LIN {X 0.078,Y -147.268,Z 1124.913,A 0.000,B 0.000,C 90.000,E1 164.393} C_DIS
LIN {X -0.047,Y -150.585,Z 1124.888,A 0.000,B 0.000,C 90.000,E1 159.880} C_DIS
LIN {X 0.032,Y -154.056,Z 1124.868,A 0.000,B 0.000,C 90.000,E1 156.230} C_DIS
LIN {X -0.042,Y -157.475,Z 1124.848,A 0.000,B 0.000,C 90.000,E1 152.666} C_DIS
LIN {X 0.044,Y -161.698,Z 1124.828,A 0.000,B 0.000,C 90.000,E1 149.076} C_DIS
LIN {X -0.078,Y -165.893,Z 1124.809,A 0.000,B 0.000,C 90.000,E1 145.595} C_DIS
LIN {X 0.047,Y -170.875,Z 1124.789,A 0.000,B 0.000,C 90.000,E1 142.065} C_DIS
LIN {X 0.075,Y -175.743,Z 1124.770,A 0.000,B 0.000,C 90.000,E1 138.609} C_DIS
LIN {X -0.052,Y -181.354,Z 1124.751,A 0.000,B 0.000,C 90.000,E1 135.243} C_DIS
LIN {X 0.081,Y -186.844,Z 1124.733,A 0.000,B 0.000,C 90.000,E1 131.838} C_DIS
LIN {X 0.035,Y -191.431,Z 1124.719,A 0.000,B 0.000,C 90.000,E1 129.358} C_DIS
LIN {X -0.032,Y -197.282,Z 1124.700,A 0.000,B 0.000,C 90.000,E1 126.091} C_DIS
LIN {X 0.094,Y -200.751,Z 1124.691,A 0.000,B 0.000,C 90.000,E1 124.326} C_DIS
LIN {X 0.093,Y -309.580,Z 1124.691,A 0.000,B 0.000,C 90.000,E1 124.326} C_DIS
LIN {X -0.009,Y -310.783,Z 1124.691,A 0.000,B 0.000,C 90.000,E1 124.326} C_DIS
LIN {X 0.192,Y -314.940,Z 1124.690,A 0.000,B 0.000,C 90.000,E1 124.119} C_DIS
LIN {X -0.044,Y -317.242,Z 1124.689,A 0.000,B 0.000,C 90.000,E1 123.992} C_DIS
LIN {X -0.078,Y -320.395,Z 1124.687,A 0.000,B 0.000,C 90.000,E1 123.658} C_DIS
LIN {X -0.134,Y -322.373,Z 1124.685,A 0.000,B 0.000,C 90.000,E1 123.372} C_DIS
LIN {X 0.082,Y -323.924,Z 1124.684,A 0.000,B 0.000,C 90.000,E1 123.038} C_DIS
LIN {X -0.010,Y -326.368,Z 1124.680,A 0.000,B 0.000,C 90.000,E1 122.418} C_DIS
LIN {X 0.001,Y -337.171,Z 1124.664,A 0.000,B 0.000,C 90.000,E1 119.589} C_DIS
LIN {X -0.050,Y -349.350,Z 1124.649,A 0.000,B 0.000,C 90.000,E1 116.821} C_DIS
LIN {X 0.109,Y -363.007,Z 1124.634,A 0.000,B 0.000,C 90.000,E1 114.079} C_DIS
LIN {X 0.104,Y -376.488,Z 1124.621,A 0.000,B 0.000,C 90.000,E1 111.716} C_DIS
LIN {X 0.164,Y -391.330,Z 1124.608,A 0.000,B 0.000,C 90.000,E1 109.396} C_DIS
LIN {X -0.034,Y -407.636,Z 1124.595,A 0.000,B 0.000,C 90.000,E1 107.166} C_DIS
LIN {X 0.043,Y -425.524,Z 1124.583,A 0.000,B 0.000,C 90.000,E1 104.954} C_DIS
LIN {X 0.016,Y -444.998,Z 1124.571,A 0.000,B 0.000,C 90.000,E1 102.827} C_DIS
LIN {X 0.148,Y -465.243,Z 1124.560,A 0.000,B 0.000,C 90.000,E1 100.838} C_DIS
LIN {X 0.147,Y -467.826,Z 1124.559,A 0.000,B 0.000,C 90.000,E1 100.602} C_DIS
LIN {X 0.183,Y -470.038,Z 1124.558,A 0.000,B 0.000,C 90.000,E1 100.366} C_DIS
LIN {X 0.135,Y -471.709,Z 1124.556,A 0.000,B 0.000,C 90.000,E1 100.141} C_DIS
LIN {X -0.008,Y -473.101,Z 1124.555,A 0.000,B 0.000,C 90.000,E1 99.905} C_DIS
LIN {X -0.154,Y -474.134,Z 1124.554,A 0.000,B 0.000,C 90.000,E1 99.670} C_DIS
LIN {X -0.038,Y -475.327,Z 1124.551,A 0.000,B 0.000,C 90.000,E1 99.151} C_DIS
LIN {X 0.158,Y -475.518,Z 1124.548,A 0.000,B 0.000,C 90.000,E1 98.624} C_DIS
LIN {X -0.181,Y -474.740,Z 1124.545,A 0.000,B 0.000,C 90.000,E1 98.163} C_DIS
LIN {X -0.048,Y -472.867,Z 1124.542,A 0.000,B 0.000,C 90.000,E1 97.644} C_DIS
LIN {X -0.186,Y -471.408,Z 1124.541,A 0.000,B 0.000,C 90.000,E1 97.409} C_DIS
LIN {X -0.064,Y -455.155,Z 1124.528,A 0.000,B 0.000,C 90.000,E1 95.106} C_DIS
LIN {X -0.132,Y -441.016,Z 1124.517,A 0.000,B 0.000,C 90.000,E1 93.037} C_DIS
LIN {X 0.012,Y -426.343,Z 1124.504,A 0.000,B 0.000,C 90.000,E1 90.630} C_DIS
LIN {X 0.187,Y -412.584,Z 1124.490,A 0.000,B 0.000,C 90.000,E1 88.167} C_DIS
LIN {X -0.140,Y -403.696,Z 1124.481,A 0.000,B 0.000,C 90.000,E1 86.560} C_DIS
LIN {X -0.185,Y -393.159,Z 1124.470,A 0.000,B 0.000,C 90.000,E1 84.609} C_DIS
LIN {X 0.011,Y -382.701,Z 1124.459,A 0.000,B 0.000,C 90.000,E1 82.591} C_DIS
LIN {X 0.081,Y -373.658,Z 1124.449,A 0.000,B 0.000,C 90.000,E1 80.849} C_DIS
LIN {X -0.009,Y -364.263,Z 1124.439,A 0.000,B 0.000,C 90.000,E1 79.106} C_DIS
LIN {X -0.200,Y -354.498,Z 1124.430,A 0.000,B 0.000,C 90.000,E1 77.353} C_DIS
LIN {X -0.144,Y -342.981,Z 1124.418,A 0.000,B 0.000,C 90.000,E1 75.227} C_DIS
LIN {X 0.050,Y -329.902,Z 1124.404,A 0.000,B 0.000,C 90.000,E1 72.725} C_DIS
LIN {X -0.017,Y -314.350,Z 1124.386,A 0.000,B 0.000,C 90.000,E1 69.571} C_DIS
LIN {X 0.067,Y -299.831,Z 1124.368,A 0.000,B 0.000,C 90.000,E1 66.305} C_DIS
LIN {X 0.084,Y -288.803,Z 1124.354,A 0.000,B 0.000,C 90.000,E1 63.640} C_DIS
LIN {X 0.089,Y -278.065,Z 1124.339,A 0.000,B 0.000,C 90.000,E1 60.923} C_DIS
LIN {X -0.064,Y -269.002,Z 1124.325,A 0.000,B 0.000,C 90.000,E1 58.535} C_DIS
LIN {X 0.071,Y -256.550,Z 1124.306,A 0.000,B 0.000,C 90.000,E1 54.975} C_DIS
LIN {X -0.011,Y -245.997,Z 1124.287,A 0.000,B 0.000,C 90.000,E1 51.743} C_DIS
LIN {X 0.089,Y -236.309,Z 1124.269,A 0.000,B 0.000,C 90.000,E1 48.405} C_DIS
LIN {X 0.096,Y -228.271,Z 1124.252,A 0.000,B 0.000,C 90.000,E1 45.405} C_DIS
LIN {X 0.063,Y -220.623,Z 1124.235,A 0.000,B 0.000,C 90.000,E1 42.366} C_DIS
LIN {X 0.036,Y -213.340,Z 1124.218,A 0.000,B 0.000,C 90.000,E1 39.277} C_DIS
LIN {X 0.023,Y -206.482,Z 1124.201,A 0.000,B 0.000,C 90.000,E1 36.137} C_DIS
LIN {X -0.021,Y -200.095,Z 1124.183,A 0.000,B 0.000,C 90.000,E1 32.959} C_DIS
LIN {X -0.089,Y -194.301,Z 1124.165,A 0.000,B 0.000,C 90.000,E1 29.745} C_DIS
LIN {X 0.018,Y -189.100,Z 1124.147,A 0.000,B 0.000,C 90.000,E1 26.437} C_DIS
LIN {X -0.007,Y -184.527,Z 1124.129,A 0.000,B 0.000,C 90.000,E1 23.131} C_DIS
LIN {X -0.066,Y -179.757,Z 1124.105,A 0.000,B 0.000,C 90.000,E1 18.960} C_DIS
LIN {X -0.036,Y -175.995,Z 1124.082,A 0.000,B 0.000,C 90.000,E1 14.717} C_DIS
LIN {X 0.069,Y -172.856,Z 1124.053,A 0.000,B 0.000,C 90.000,E1 9.557} C_DIS
LIN {X -0.002,Y -170.940,Z 1124.010,A 0.000,B 0.000,C 90.000,E1 1.835} C_DIS
LIN {X -0.050,Y -172.525,Z 1123.964,A 0.000,B 0.000,C 90.000,E1 353.514} C_DIS
LIN {X 0.020,Y -175.335,Z 1123.935,A 0.000,B 0.000,C 90.000,E1 348.342} C_DIS
LIN {X -0.052,Y -178.751,Z 1123.912,A 0.000,B 0.000,C 90.000,E1 344.102} C_DIS
LIN {X -0.072,Y -183.004,Z 1123.888,A 0.000,B 0.000,C 90.000,E1 339.880} C_DIS
LIN {X 0.066,Y -187.097,Z 1123.870,A 0.000,B 0.000,C 90.000,E1 336.485} C_DIS
LIN {X 0.023,Y -191.887,Z 1123.851,A 0.000,B 0.000,C 90.000,E1 333.179} C_DIS
LIN {X -0.066,Y -197.332,Z 1123.833,A 0.000,B 0.000,C 90.000,E1 329.921} C_DIS
LIN {X 0.107,Y -203.385,Z 1123.815,A 0.000,B 0.000,C 90.000,E1 326.628} C_DIS
LIN {X -0.018,Y -210.290,Z 1123.797,A 0.000,B 0.000,C 90.000,E1 323.463} C_DIS
LIN {X 0.116,Y -217.935,Z 1123.779,A 0.000,B 0.000,C 90.000,E1 320.275} C_DIS
LIN {X -0.067,Y -226.470,Z 1123.762,A 0.000,B 0.000,C 90.000,E1 317.229} C_DIS
LIN {X -0.061,Y -236.018,Z 1123.745,A 0.000,B 0.000,C 90.000,E1 314.190} C_DIS
LIN {X 0.073,Y -243.903,Z 1123.733,A 0.000,B 0.000,C 90.000,E1 311.919} C_DIS
LIN {X 0.075,Y -255.655,Z 1123.717,A 0.000,B 0.000,C 90.000,E1 308.991} C_DIS
LIN {X -0.061,Y -265.510,Z 1123.705,A 0.000,B 0.000,C 90.000,E1 306.870} C_DIS
LIN {X 0.065,Y -279.774,Z 1123.689,A 0.000,B 0.000,C 90.000,E1 304.040} C_DIS
LIN {X -0.065,Y -294.990,Z 1123.674,A 0.000,B 0.000,C 90.000,E1 301.337} C_DIS
LIN {X -0.059,Y -314.165,Z 1123.657,A 0.000,B 0.000,C 90.000,E1 298.359} C_DIS
LIN {X -0.007,Y -330.283,Z 1123.645,A 0.000,B 0.000,C 90.000,E1 296.104} C_DIS
LIN {X -0.108,Y -345.206,Z 1123.635,A 0.000,B 0.000,C 90.000,E1 294.259} C_DIS
LIN {X 0.181,Y -358.205,Z 1123.627,A 0.000,B 0.000,C 90.000,E1 292.770} C_DIS
LIN {X -0.036,Y -371.604,Z 1123.619,A 0.000,B 0.000,C 90.000,E1 291.461} C_DIS
LIN {X -0.066,Y -393.675,Z 1123.608,A 0.000,B 0.000,C 90.000,E1 289.450} C_DIS
LIN {X -0.014,Y -404.411,Z 1123.603,A 0.000,B 0.000,C 90.000,E1 288.489} C_DIS
LIN {X -0.010,Y -414.928,Z 1123.597,A 0.000,B 0.000,C 90.000,E1 287.511} C_DIS
LIN {X 0.218,Y -422.666,Z 1123.593,A 0.000,B 0.000,C 90.000,E1 286.732} C_DIS
LIN {X -0.221,Y -430.176,Z 1123.589,A 0.000,B 0.000,C 90.000,E1 286.024} C_DIS
LIN {X 0.112,Y -437.408,Z 1123.584,A 0.000,B 0.000,C 90.000,E1 285.190} C_DIS
LIN {X -0.030,Y -444.251,Z 1123.580,A 0.000,B 0.000,C 90.000,E1 284.411} C_DIS
LIN {X 0.216,Y -450.480,Z 1123.576,A 0.000,B 0.000,C 90.000,E1 283.592} C_DIS
LIN {X -0.174,Y -454.313,Z 1123.573,A 0.000,B 0.000,C 90.000,E1 283.119} C_DIS
LIN {X 0.165,Y -459.376,Z 1123.568,A 0.000,B 0.000,C 90.000,E1 282.299} C_DIS
LIN {X 0.107,Y -463.742,Z 1123.564,A 0.000,B 0.000,C 90.000,E1 281.535} C_DIS
LIN {X -0.159,Y -468.724,Z 1123.558,A 0.000,B 0.000,C 90.000,E1 280.546} C_DIS
LIN {X -0.147,Y -471.821,Z 1123.554,A 0.000,B 0.000,C 90.000,E1 279.782} C_DIS
LIN {X -0.053,Y -473.578,Z 1123.551,A 0.000,B 0.000,C 90.000,E1 279.265} C_DIS
LIN {X 0.057,Y -474.975,Z 1123.549,A 0.000,B 0.000,C 90.000,E1 278.746} C_DIS
LIN {X 0.249,Y -476.177,Z 1123.546,A 0.000,B 0.000,C 90.000,E1 278.219} C_DIS
LIN {X -0.093,Y -477.066,Z 1123.543,A 0.000,B 0.000,C 90.000,E1 277.757} C_DIS
LIN {X 0.046,Y -477.654,Z 1123.540,A 0.000,B 0.000,C 90.000,E1 277.239} C_DIS
LIN {X 0.191,Y -477.940,Z 1123.537,A 0.000,B 0.000,C 90.000,E1 276.720} C_DIS
LIN {X -0.135,Y -477.901,Z 1123.535,A 0.000,B 0.000,C 90.000,E1 276.258} C_DIS
LIN {X 0.015,Y -477.520,Z 1123.532,A 0.000,B 0.000,C 90.000,E1 275.739} C_DIS
LIN {X 0.163,Y -476.836,Z 1123.529,A 0.000,B 0.000,C 90.000,E1 275.220} C_DIS
LIN {X -0.167,Y -475.804,Z 1123.526,A 0.000,B 0.000,C 90.000,E1 274.759} C_DIS
LIN {X -0.063,Y -474.319,Z 1123.524,A 0.000,B 0.000,C 90.000,E1 274.245} C_DIS
LIN {X 0.069,Y -472.342,Z 1123.521,A 0.000,B 0.000,C 90.000,E1 273.726} C_DIS
LIN {X -0.119,Y -471.140,Z 1123.519,A 0.000,B 0.000,C 90.000,E1 273.498} C_DIS
LIN {X -0.007,Y -468.090,Z 1123.517,A 0.000,B 0.000,C 90.000,E1 272.980} C_DIS
LIN {X -0.202,Y -466.283,Z 1123.515,A 0.000,B 0.000,C 90.000,E1 272.751} C_DIS
LIN {X -0.140,Y -461.786,Z 1123.512,A 0.000,B 0.000,C 90.000,E1 272.236} C_DIS
LIN {X 0.111,Y -459.021,Z 1123.511,A 0.000,B 0.000,C 90.000,E1 271.949} C_DIS
LIN {X 0.029,Y -452.897,Z 1123.508,A 0.000,B 0.000,C 90.000,E1 271.489} C_DIS
LIN {X 0.040,Y -446.345,Z 1123.506,A 0.000,B 0.000,C 90.000,E1 271.088} C_DIS
LIN {X 0.084,Y -439.442,Z 1123.504,A 0.000,B 0.000,C 90.000,E1 270.745} C_DIS
LIN {X 0.121,Y -432.411,Z 1123.503,A 0.000,B 0.000,C 90.000,E1 270.458} C_DIS
LIN {X 0.079,Y -425.348,Z 1123.501,A 0.000,B 0.000,C 90.000,E1 270.229} C_DIS
LIN {X -0.107,Y -418.092,Z 1123.500,A 0.000,B 0.000,C 90.000,E1 270.057} C_DIS
LIN {X -0.044,Y -410.673,Z 1123.499,A 0.000,B 0.000,C 90.000,E1 269.885} C_DIS
LIN {X -0.162,Y -403.059,Z 1123.499,A 0.000,B 0.000,C 90.000,E1 269.771} C_DIS
LIN {X -0.080,Y -393.478,Z 1123.498,A 0.000,B 0.000,C 90.000,E1 269.656} C_DIS
LIN {X 0.007,Y -384.032,Z 1123.498,A 0.000,B 0.000,C 90.000,E1 269.599} C_DIS
LIN {X -0.019,Y -181.463,Z 1123.498,A 0.000,B 0.000,C 90.000,E1 269.599} C_DIS
LIN {X -0.068,Y -180.906,Z 1123.474,A 0.000,B 0.000,C 90.000,E1 265.355} C_DIS
LIN {X 0.006,Y -180.671,Z 1123.469,A 0.000,B 0.000,C 90.000,E1 264.489} C_DIS
LIN {X 0.080,Y -178.752,Z 1123.441,A 0.000,B 0.000,C 90.000,E1 259.398} C_DIS
LIN {X -0.022,Y -175.799,Z 1123.413,A 0.000,B 0.000,C 90.000,E1 254.338} C_DIS
LIN {X -0.028,Y -171.985,Z 1123.384,A 0.000,B 0.000,C 90.000,E1 249.209} C_DIS
LIN {X 0.010,Y -171.391,Z 1123.380,A 0.000,B 0.000,C 90.000,E1 248.337} C_DIS
LIN {X -0.004,Y -167.634,Z 1123.356,A 0.000,B 0.000,C 90.000,E1 244.024} C_DIS
LIN {X 0.010,Y -166.292,Z 1123.346,A 0.000,B 0.000,C 90.000,E1 242.281} C_DIS
LIN {X 0.004,Y -163.039,Z 1123.327,A 0.000,B 0.000,C 90.000,E1 238.791} C_DIS
LIN {X -0.034,Y -160.970,Z 1123.312,A 0.000,B 0.000,C 90.000,E1 236.167} C_DIS
LIN {X -0.056,Y -157.722,Z 1123.292,A 0.000,B 0.000,C 90.000,E1 232.637} C_DIS
LIN {X 0.103,Y -155.762,Z 1123.277,A 0.000,B 0.000,C 90.000,E1 229.908} C_DIS
LIN {X -0.060,Y -152.017,Z 1123.253,A 0.000,B 0.000,C 90.000,E1 225.486} C_DIS
LIN {X -0.043,Y -150.264,Z 1123.238,A 0.000,B 0.000,C 90.000,E1 222.771} C_DIS
LIN {X -0.024,Y -147.017,Z 1123.212,A 0.000,B 0.000,C 90.000,E1 218.222} C_DIS
LIN {X -0.003,Y -145.600,Z 1123.197,A 0.000,B 0.000,C 90.000,E1 215.471} C_DIS
LIN {X 0.001,Y -142.986,Z 1123.172,A 0.000,B 0.000,C 90.000,E1 210.875} C_DIS
LIN {X 0.000,Y -141.613,Z 1123.151,A 0.000,B 0.000,C 90.000,E1 207.180} C_DIS
LIN {X 0.042,Y -139.428,Z 1123.115,A 0.000,B 0.000,C 90.000,E1 200.663} C_DIS
LIN {X -0.038,Y -139.158,Z 1123.104,A 0.000,B 0.000,C 90.000,E1 198.833} C_DIS
LIN {X -0.022,Y -138.343,Z 1123.058,A 0.000,B 0.000,C 90.000,E1 190.423} C_DIS
LIN {X -0.039,Y -139.481,Z 1123.006,A 0.000,B 0.000,C 90.000,E1 181.088} C_DIS
LIN {X 0.041,Y -141.072,Z 1122.975,A 0.000,B 0.000,C 90.000,E1 175.469} C_DIS
LIN {X -0.004,Y -142.447,Z 1122.959,A 0.000,B 0.000,C 90.000,E1 172.704} C_DIS
LIN {X -0.056,Y -144.687,Z 1122.934,A 0.000,B 0.000,C 90.000,E1 168.105} C_DIS
LIN {X 0.039,Y -147.280,Z 1122.913,A 0.000,B 0.000,C 90.000,E1 164.393} C_DIS
LIN {X 0.054,Y -150.598,Z 1122.888,A 0.000,B 0.000,C 90.000,E1 159.826} C_DIS
LIN {X -0.009,Y -154.071,Z 1122.868,A 0.000,B 0.000,C 90.000,E1 156.230} C_DIS
LIN {X 0.057,Y -157.491,Z 1122.848,A 0.000,B 0.000,C 90.000,E1 152.615} C_DIS
LIN {X 0.003,Y -161.717,Z 1122.828,A 0.000,B 0.000,C 90.000,E1 149.076} C_DIS
LIN {X 0.017,Y -165.911,Z 1122.809,A 0.000,B 0.000,C 90.000,E1 145.548} C_DIS
LIN {X 0.004,Y -170.897,Z 1122.789,A 0.000,B 0.000,C 90.000,E1 142.065} C_DIS
LIN {X 0.030,Y -175.765,Z 1122.770,A 0.000,B 0.000,C 90.000,E1 138.609} C_DIS
LIN {X -0.097,Y -181.375,Z 1122.751,A 0.000,B 0.000,C 90.000,E1 135.243} C_DIS
LIN {X 0.036,Y -186.870,Z 1122.733,A 0.000,B 0.000,C 90.000,E1 131.838} C_DIS
LIN {X -0.011,Y -191.454,Z 1122.719,A 0.000,B 0.000,C 90.000,E1 129.358} C_DIS
LIN {X -0.079,Y -197.308,Z 1122.700,A 0.000,B 0.000,C 90.000,E1 126.091} C_DIS
LIN {X -0.073,Y -200.691,Z 1122.691,A 0.000,B 0.000,C 90.000,E1 124.405} C_DIS
LIN {X -0.165,Y -309.271,Z 1122.691,A 0.000,B 0.000,C 90.000,E1 124.405} C_DIS
LIN {X -0.054,Y -314.738,Z 1122.690,A 0.000,B 0.000,C 90.000,E1 124.199} C_DIS
LIN {X 0.059,Y -317.249,Z 1122.689,A 0.000,B 0.000,C 90.000,E1 123.992} C_DIS
LIN {X 0.024,Y -320.601,Z 1122.687,A 0.000,B 0.000,C 90.000,E1 123.627} C_DIS
LIN {X 0.202,Y -322.540,Z 1122.685,A 0.000,B 0.000,C 90.000,E1 123.293} C_DIS
LIN {X -0.066,Y -324.057,Z 1122.683,A 0.000,B 0.000,C 90.000,E1 123.038} C_DIS
LIN {X -0.128,Y -329.897,Z 1122.675,A 0.000,B 0.000,C 90.000,E1 121.465} C_DIS
LIN {X 0.100,Y -341.161,Z 1122.659,A 0.000,B 0.000,C 90.000,E1 118.615} C_DIS
LIN {X 0.176,Y -353.831,Z 1122.644,A 0.000,B 0.000,C 90.000,E1 115.848} C_DIS
LIN {X -0.176,Y -368.026,Z 1122.629,A 0.000,B 0.000,C 90.000,E1 113.206} C_DIS
LIN {X -0.068,Y -382.020,Z 1122.616,A 0.000,B 0.000,C 90.000,E1 110.844} C_DIS
LIN {X -0.012,Y -397.413,Z 1122.603,A 0.000,B 0.000,C 90.000,E1 108.544} C_DIS
LIN {X -0.074,Y -414.315,Z 1122.591,A 0.000,B 0.000,C 90.000,E1 106.315} C_DIS
LIN {X 0.045,Y -432.847,Z 1122.578,A 0.000,B 0.000,C 90.000,E1 104.120} C_DIS
LIN {X -0.125,Y -452.724,Z 1122.567,A 0.000,B 0.000,C 90.000,E1 102.063} C_DIS
LIN {X -0.017,Y -468.016,Z 1122.559,A 0.000,B 0.000,C 90.000,E1 100.602} C_DIS
LIN {X -0.007,Y -470.194,Z 1122.558,A 0.000,B 0.000,C 90.000,E1 100.366} C_DIS
LIN {X -0.082,Y -471.839,Z 1122.556,A 0.000,B 0.000,C 90.000,E1 100.141} C_DIS
LIN {X -0.226,Y -473.187,Z 1122.555,A 0.000,B 0.000,C 90.000,E1 99.905} C_DIS
LIN {X 0.096,Y -474.185,Z 1122.553,A 0.000,B 0.000,C 90.000,E1 99.613} C_DIS
LIN {X -0.256,Y -475.321,Z 1122.551,A 0.000,B 0.000,C 90.000,E1 99.151} C_DIS
LIN {X -0.060,Y -475.460,Z 1122.548,A 0.000,B 0.000,C 90.000,E1 98.624} C_DIS
LIN {X 0.072,Y -474.628,Z 1122.545,A 0.000,B 0.000,C 90.000,E1 98.106} C_DIS
LIN {X 0.204,Y -472.688,Z 1122.542,A 0.000,B 0.000,C 90.000,E1 97.587} C_DIS
LIN {X 0.065,Y -471.185,Z 1122.541,A 0.000,B 0.000,C 90.000,E1 97.352} C_DIS
LIN {X 0.175,Y -454.915,Z 1122.528,A 0.000,B 0.000,C 90.000,E1 95.049} C_DIS
LIN {X 0.095,Y -440.803,Z 1122.517,A 0.000,B 0.000,C 90.000,E1 92.980} C_DIS
LIN {X -0.200,Y -426.134,Z 1122.503,A 0.000,B 0.000,C 90.000,E1 90.630} C_DIS
LIN {X -0.010,Y -412.392,Z 1122.490,A 0.000,B 0.000,C 90.000,E1 88.165} C_DIS
LIN {X 0.054,Y -403.476,Z 1122.481,A 0.000,B 0.000,C 90.000,E1 86.502} C_DIS
LIN {X 0.037,Y -392.943,Z 1122.470,A 0.000,B 0.000,C 90.000,E1 84.546} C_DIS
LIN {X -0.196,Y -382.457,Z 1122.459,A 0.000,B 0.000,C 90.000,E1 82.591} C_DIS
LIN {X -0.125,Y -373.410,Z 1122.449,A 0.000,B 0.000,C 90.000,E1 80.849} C_DIS
LIN {X 0.143,Y -363.997,Z 1122.439,A 0.000,B 0.000,C 90.000,E1 79.050} C_DIS
LIN {X 0.020,Y -354.232,Z 1122.429,A 0.000,B 0.000,C 90.000,E1 77.285} C_DIS
LIN {X -0.016,Y -342.704,Z 1122.418,A 0.000,B 0.000,C 90.000,E1 75.172} C_DIS
LIN {X -0.153,Y -329.628,Z 1122.404,A 0.000,B 0.000,C 90.000,E1 72.725} C_DIS
LIN {X 0.076,Y -314.071,Z 1122.386,A 0.000,B 0.000,C 90.000,E1 69.518} C_DIS
LIN {X -0.023,Y -301.005,Z 1122.370,A 0.000,B 0.000,C 90.000,E1 66.613} C_DIS
LIN {X -0.114,Y -288.562,Z 1122.353,A 0.000,B 0.000,C 90.000,E1 63.640} C_DIS
LIN {X 0.090,Y -276.514,Z 1122.336,A 0.000,B 0.000,C 90.000,E1 60.539} C_DIS
LIN {X 0.037,Y -267.447,Z 1122.323,A 0.000,B 0.000,C 90.000,E1 58.122} C_DIS
LIN {X -0.123,Y -256.262,Z 1122.305,A 0.000,B 0.000,C 90.000,E1 54.975} C_DIS
LIN {X -0.012,Y -245.726,Z 1122.287,A 0.000,B 0.000,C 90.000,E1 51.698} C_DIS
LIN {X -0.111,Y -235.996,Z 1122.269,A 0.000,B 0.000,C 90.000,E1 48.405} C_DIS
LIN {X -0.106,Y -227.948,Z 1122.252,A 0.000,B 0.000,C 90.000,E1 45.405} C_DIS
LIN {X 0.023,Y -220.291,Z 1122.235,A 0.000,B 0.000,C 90.000,E1 42.324} C_DIS
LIN {X 0.131,Y -212.976,Z 1122.218,A 0.000,B 0.000,C 90.000,E1 39.197} C_DIS
LIN {X -0.017,Y -206.098,Z 1122.200,A 0.000,B 0.000,C 90.000,E1 36.091} C_DIS
LIN {X 0.046,Y -199.720,Z 1122.183,A 0.000,B 0.000,C 90.000,E1 32.880} C_DIS
LIN {X -0.036,Y -193.939,Z 1122.165,A 0.000,B 0.000,C 90.000,E1 29.667} C_DIS
LIN {X 0.056,Y -188.733,Z 1122.146,A 0.000,B 0.000,C 90.000,E1 26.360} C_DIS
LIN {X -0.056,Y -184.163,Z 1122.128,A 0.000,B 0.000,C 90.000,E1 23.078} C_DIS
LIN {X 0.020,Y -180.266,Z 1122.109,A 0.000,B 0.000,C 90.000,E1 19.704} C_DIS
LIN {X 0.000,Y -176.334,Z 1122.086,A 0.000,B 0.000,C 90.000,E1 15.481} C_DIS
LIN {X 0.087,Y -173.408,Z 1122.062,A 0.000,B 0.000,C 90.000,E1 11.186} C_DIS
LIN {X -0.060,Y -171.090,Z 1122.029,A 0.000,B 0.000,C 90.000,E1 5.220} C_DIS
LIN {X -0.062,Y -172.230,Z 1121.964,A 0.000,B 0.000,C 90.000,E1 353.514} C_DIS
LIN {X -0.004,Y -175.013,Z 1121.935,A 0.000,B 0.000,C 90.000,E1 348.342} C_DIS
LIN {X -0.086,Y -178.430,Z 1121.911,A 0.000,B 0.000,C 90.000,E1 344.102} C_DIS
LIN {X 0.055,Y -182.673,Z 1121.888,A 0.000,B 0.000,C 90.000,E1 339.826} C_DIS
LIN {X 0.011,Y -186.756,Z 1121.869,A 0.000,B 0.000,C 90.000,E1 336.485} C_DIS
LIN {X -0.040,Y -191.571,Z 1121.851,A 0.000,B 0.000,C 90.000,E1 333.179} C_DIS
LIN {X 0.030,Y -197.013,Z 1121.833,A 0.000,B 0.000,C 90.000,E1 329.871} C_DIS
LIN {X 0.022,Y -203.098,Z 1121.815,A 0.000,B 0.000,C 90.000,E1 326.628} C_DIS
LIN {X 0.056,Y -210.032,Z 1121.797,A 0.000,B 0.000,C 90.000,E1 323.417} C_DIS
LIN {X 0.012,Y -217.714,Z 1121.779,A 0.000,B 0.000,C 90.000,E1 320.275} C_DIS
LIN {X -0.015,Y -226.272,Z 1121.762,A 0.000,B 0.000,C 90.000,E1 317.187} C_DIS
LIN {X -0.062,Y -237.098,Z 1121.743,A 0.000,B 0.000,C 90.000,E1 313.785} C_DIS
LIN {X 0.080,Y -246.590,Z 1121.729,A 0.000,B 0.000,C 90.000,E1 311.148} C_DIS
LIN {X -0.066,Y -255.540,Z 1121.717,A 0.000,B 0.000,C 90.000,E1 308.991} C_DIS
LIN {X 0.062,Y -267.220,Z 1121.703,A 0.000,B 0.000,C 90.000,E1 306.457} C_DIS
LIN {X 0.192,Y -283.502,Z 1121.685,A 0.000,B 0.000,C 90.000,E1 303.293} C_DIS
LIN {X 0.176,Y -295.064,Z 1121.674,A 0.000,B 0.000,C 90.000,E1 301.258} C_DIS
LIN {X 0.045,Y -314.270,Z 1121.657,A 0.000,B 0.000,C 90.000,E1 298.309} C_DIS
LIN {X 0.110,Y -330.421,Z 1121.645,A 0.000,B 0.000,C 90.000,E1 296.052} C_DIS
LIN {X -0.057,Y -345.496,Z 1121.634,A 0.000,B 0.000,C 90.000,E1 294.207} C_DIS
LIN {X -0.032,Y -358.397,Z 1121.626,A 0.000,B 0.000,C 90.000,E1 292.770} C_DIS
LIN {X 0.031,Y -371.910,Z 1121.619,A 0.000,B 0.000,C 90.000,E1 291.408} C_DIS
LIN {X 0.077,Y -393.919,Z 1121.608,A 0.000,B 0.000,C 90.000,E1 289.396} C_DIS
LIN {X 0.204,Y -404.741,Z 1121.602,A 0.000,B 0.000,C 90.000,E1 288.417} C_DIS
LIN {X 0.073,Y -415.316,Z 1121.597,A 0.000,B 0.000,C 90.000,E1 287.457} C_DIS
LIN {X -0.163,Y -425.497,Z 1121.592,A 0.000,B 0.000,C 90.000,E1 286.496} C_DIS
LIN {X -0.139,Y -432.945,Z 1121.587,A 0.000,B 0.000,C 90.000,E1 285.717} C_DIS
LIN {X 0.026,Y -440.074,Z 1121.583,A 0.000,B 0.000,C 90.000,E1 284.898} C_DIS
LIN {X -0.088,Y -446.728,Z 1121.578,A 0.000,B 0.000,C 90.000,E1 284.120} C_DIS
LIN {X 0.177,Y -452.784,Z 1121.574,A 0.000,B 0.000,C 90.000,E1 283.300} C_DIS
LIN {X 0.066,Y -458.094,Z 1121.570,A 0.000,B 0.000,C 90.000,E1 282.535} C_DIS
LIN {X -0.007,Y -462.671,Z 1121.565,A 0.000,B 0.000,C 90.000,E1 281.771} C_DIS
LIN {X -0.039,Y -466.670,Z 1121.561,A 0.000,B 0.000,C 90.000,E1 281.007} C_DIS
LIN {X -0.129,Y -470.136,Z 1121.557,A 0.000,B 0.000,C 90.000,E1 280.254} C_DIS
LIN {X 0.041,Y -472.123,Z 1121.554,A 0.000,B 0.000,C 90.000,E1 279.726} C_DIS
LIN {X 0.138,Y -473.867,Z 1121.551,A 0.000,B 0.000,C 90.000,E1 279.208} C_DIS
LIN {X -0.219,Y -475.302,Z 1121.548,A 0.000,B 0.000,C 90.000,E1 278.746} C_DIS
LIN {X -0.025,Y -476.432,Z 1121.546,A 0.000,B 0.000,C 90.000,E1 278.219} C_DIS
LIN {X 0.107,Y -477.330,Z 1121.543,A 0.000,B 0.000,C 90.000,E1 277.701} C_DIS
LIN {X -0.226,Y -477.922,Z 1121.540,A 0.000,B 0.000,C 90.000,E1 277.239} C_DIS
LIN {X -0.079,Y -478.150,Z 1121.537,A 0.000,B 0.000,C 90.000,E1 276.720} C_DIS
LIN {X 0.071,Y -478.155,Z 1121.535,A 0.000,B 0.000,C 90.000,E1 276.201} C_DIS
LIN {X 0.222,Y -477.778,Z 1121.532,A 0.000,B 0.000,C 90.000,E1 275.682} C_DIS
LIN {X -0.103,Y -477.099,Z 1121.529,A 0.000,B 0.000,C 90.000,E1 275.220} C_DIS
LIN {X 0.044,Y -476.033,Z 1121.526,A 0.000,B 0.000,C 90.000,E1 274.702} C_DIS
LIN {X 0.148,Y -474.584,Z 1121.523,A 0.000,B 0.000,C 90.000,E1 274.188} C_DIS
LIN {X -0.190,Y -472.549,Z 1121.521,A 0.000,B 0.000,C 90.000,E1 273.726} C_DIS
LIN {X 0.094,Y -471.347,Z 1121.519,A 0.000,B 0.000,C 90.000,E1 273.440} C_DIS
LIN {X 0.205,Y -468.299,Z 1121.516,A 0.000,B 0.000,C 90.000,E1 272.922} C_DIS
LIN {X -0.191,Y -464.324,Z 1121.514,A 0.000,B 0.000,C 90.000,E1 272.465} C_DIS
LIN {X 0.073,Y -461.961,Z 1121.512,A 0.000,B 0.000,C 90.000,E1 272.178} C_DIS
LIN {X -0.137,Y -459.178,Z 1121.511,A 0.000,B 0.000,C 90.000,E1 271.949} C_DIS
LIN {X 0.214,Y -453.034,Z 1121.508,A 0.000,B 0.000,C 90.000,E1 271.432} C_DIS
LIN {X 0.206,Y -446.431,Z 1121.506,A 0.000,B 0.000,C 90.000,E1 271.031} C_DIS
LIN {X -0.171,Y -439.514,Z 1121.504,A 0.000,B 0.000,C 90.000,E1 270.745} C_DIS
LIN {X -0.096,Y -432.594,Z 1121.502,A 0.000,B 0.000,C 90.000,E1 270.458} C_DIS
LIN {X -0.104,Y -425.559,Z 1121.501,A 0.000,B 0.000,C 90.000,E1 270.229} C_DIS
LIN {X 0.143,Y -418.405,Z 1121.500,A 0.000,B 0.000,C 90.000,E1 270.000} C_DIS
LIN {X 0.204,Y -410.942,Z 1121.499,A 0.000,B 0.000,C 90.000,E1 269.828} C_DIS
LIN {X 0.083,Y -403.019,Z 1121.498,A 0.000,B 0.000,C 90.000,E1 269.714} C_DIS
LIN {X 0.157,Y -393.054,Z 1121.498,A 0.000,B 0.000,C 90.000,E1 269.599} C_DIS
LIN {X -0.073,Y -386.219,Z 1121.498,A 0.000,B 0.000,C 90.000,E1 269.599} C_DIS
LIN {X -0.070,Y -181.459,Z 1121.498,A 0.000,B 0.000,C 90.000,E1 269.599} C_DIS
LIN {X 0.053,Y -180.867,Z 1121.472,A 0.000,B 0.000,C 90.000,E1 265.008} C_DIS
LIN {X -0.070,Y -178.982,Z 1121.444,A 0.000,B 0.000,C 90.000,E1 259.982} C_DIS
LIN {X -0.058,Y -177.954,Z 1121.435,A 0.000,B 0.000,C 90.000,E1 258.285} C_DIS
LIN {X -0.039,Y -175.597,Z 1121.411,A 0.000,B 0.000,C 90.000,E1 254.031} C_DIS
LIN {X -0.026,Y -172.320,Z 1121.387,A 0.000,B 0.000,C 90.000,E1 249.752} C_DIS
LIN {X -0.047,Y -171.799,Z 1121.383,A 0.000,B 0.000,C 90.000,E1 248.901} C_DIS
LIN {X -0.010,Y -169.471,Z 1121.368,A 0.000,B 0.000,C 90.000,E1 246.305} C_DIS
LIN {X 0.046,Y -166.798,Z 1121.349,A 0.000,B 0.000,C 90.000,E1 242.820} C_DIS
LIN {X 0.041,Y -162.780,Z 1121.325,A 0.000,B 0.000,C 90.000,E1 238.456} C_DIS
LIN {X 0.016,Y -161.468,Z 1121.315,A 0.000,B 0.000,C 90.000,E1 236.707} C_DIS
LIN {X 0.057,Y -157.463,Z 1121.291,A 0.000,B 0.000,C 90.000,E1 232.271} C_DIS
LIN {X -0.010,Y -155.475,Z 1121.276,A 0.000,B 0.000,C 90.000,E1 229.622} C_DIS
LIN {X -0.077,Y -151.786,Z 1121.251,A 0.000,B 0.000,C 90.000,E1 225.162} C_DIS
LIN {X -0.063,Y -149.993,Z 1121.236,A 0.000,B 0.000,C 90.000,E1 222.447} C_DIS
LIN {X -0.032,Y -146.823,Z 1121.210,A 0.000,B 0.000,C 90.000,E1 217.890} C_DIS
LIN {X 0.074,Y -145.403,Z 1121.195,A 0.000,B 0.000,C 90.000,E1 215.105} C_DIS
LIN {X -0.009,Y -142.836,Z 1121.170,A 0.000,B 0.000,C 90.000,E1 210.541} C_DIS
LIN {X -0.078,Y -141.449,Z 1121.149,A 0.000,B 0.000,C 90.000,E1 206.873} C_DIS
LIN {X -0.039,Y -139.371,Z 1121.113,A 0.000,B 0.000,C 90.000,E1 200.355} C_DIS
LIN {X 0.036,Y -138.820,Z 1121.097,A 0.000,B 0.000,C 90.000,E1 197.528} C_DIS
LIN {X -0.007,Y -138.352,Z 1121.056,A 0.000,B 0.000,C 90.000,E1 190.074} C_DIS
LIN {X -0.035,Y -139.534,Z 1121.004,A 0.000,B 0.000,C 90.000,E1 180.745} C_DIS
LIN {X 0.058,Y -141.220,Z 1120.973,A 0.000,B 0.000,C 90.000,E1 175.122} C_DIS
LIN {X 0.017,Y -142.593,Z 1120.958,A 0.000,B 0.000,C 90.000,E1 172.356} C_DIS
LIN {X -0.029,Y -144.894,Z 1120.932,A 0.000,B 0.000,C 90.000,E1 167.757} C_DIS
LIN {X -0.076,Y -147.523,Z 1120.911,A 0.000,B 0.000,C 90.000,E1 164.102} C_DIS
LIN {X -0.002,Y -150.119,Z 1120.891,A 0.000,B 0.000,C 90.000,E1 160.423} C_DIS
LIN {X 0.010,Y -153.480,Z 1120.871,A 0.000,B 0.000,C 90.000,E1 156.794} C_DIS
LIN {X 0.074,Y -157.843,Z 1120.846,A 0.000,B 0.000,C 90.000,E1 152.281} C_DIS
LIN {X 0.029,Y -162.128,Z 1120.826,A 0.000,B 0.000,C 90.000,E1 148.742} C_DIS
LIN {X 0.010,Y -166.331,Z 1120.807,A 0.000,B 0.000,C 90.000,E1 145.229} C_DIS
LIN {X 0.016,Y -171.349,Z 1120.787,A 0.000,B 0.000,C 90.000,E1 141.743} C_DIS
LIN {X -0.057,Y -176.252,Z 1120.768,A 0.000,B 0.000,C 90.000,E1 138.324} C_DIS
LIN {X 0.062,Y -180.535,Z 1120.754,A 0.000,B 0.000,C 90.000,E1 135.729} C_DIS
LIN {X 0.041,Y -185.937,Z 1120.735,A 0.000,B 0.000,C 90.000,E1 132.366} C_DIS
LIN {X -0.024,Y -190.567,Z 1120.722,A 0.000,B 0.000,C 90.000,E1 129.886} C_DIS
LIN {X 0.007,Y -196.317,Z 1120.703,A 0.000,B 0.000,C 90.000,E1 126.583} C_DIS
LIN {X 0.027,Y -200.638,Z 1120.691,A 0.000,B 0.000,C 90.000,E1 124.405} C_DIS
LIN {X -0.005,Y -309.482,Z 1120.691,A 0.000,B 0.000,C 90.000,E1 124.405} C_DIS
LIN {X -0.025,Y -313.661,Z 1120.690,A 0.000,B 0.000,C 90.000,E1 124.278} C_DIS
LIN {X 0.132,Y -315.771,Z 1120.690,A 0.000,B 0.000,C 90.000,E1 124.119} C_DIS
LIN {X -0.096,Y -319.650,Z 1120.688,A 0.000,B 0.000,C 90.000,E1 123.785} C_DIS
LIN {X 0.056,Y -323.137,Z 1120.685,A 0.000,B 0.000,C 90.000,E1 123.214} C_DIS
LIN {X 0.137,Y -324.574,Z 1120.683,A 0.000,B 0.000,C 90.000,E1 122.880} C_DIS
LIN {X 0.048,Y -336.456,Z 1120.665,A 0.000,B 0.000,C 90.000,E1 119.745} C_DIS
LIN {X -0.160,Y -348.552,Z 1120.650,A 0.000,B 0.000,C 90.000,E1 117.001} C_DIS
LIN {X -0.036,Y -362.118,Z 1120.635,A 0.000,B 0.000,C 90.000,E1 114.259} C_DIS
LIN {X -0.074,Y -375.513,Z 1120.622,A 0.000,B 0.000,C 90.000,E1 111.897} C_DIS
LIN {X -0.048,Y -390.261,Z 1120.609,A 0.000,B 0.000,C 90.000,E1 109.577} C_DIS
LIN {X 0.227,Y -406.468,Z 1120.596,A 0.000,B 0.000,C 90.000,E1 107.275} C_DIS
LIN {X -0.242,Y -424.247,Z 1120.584,A 0.000,B 0.000,C 90.000,E1 105.134} C_DIS
LIN {X 0.200,Y -443.634,Z 1120.572,A 0.000,B 0.000,C 90.000,E1 102.939} C_DIS
LIN {X 0.241,Y -463.843,Z 1120.561,A 0.000,B 0.000,C 90.000,E1 100.950} C_DIS
LIN {X 0.169,Y -468.898,Z 1120.558,A 0.000,B 0.000,C 90.000,E1 100.489} C_DIS
LIN {X 0.196,Y -470.830,Z 1120.557,A 0.000,B 0.000,C 90.000,E1 100.254} C_DIS
LIN {X 0.049,Y -472.422,Z 1120.556,A 0.000,B 0.000,C 90.000,E1 100.018} C_DIS
LIN {X -0.180,Y -473.615,Z 1120.554,A 0.000,B 0.000,C 90.000,E1 99.792} C_DIS
LIN {X 0.010,Y -475.065,Z 1120.552,A 0.000,B 0.000,C 90.000,E1 99.265} C_DIS
LIN {X 0.130,Y -475.481,Z 1120.549,A 0.000,B 0.000,C 90.000,E1 98.746} C_DIS
LIN {X -0.140,Y -474.933,Z 1120.546,A 0.000,B 0.000,C 90.000,E1 98.276} C_DIS
LIN {X -0.008,Y -473.337,Z 1120.543,A 0.000,B 0.000,C 90.000,E1 97.757} C_DIS
LIN {X -0.208,Y -472.061,Z 1120.542,A 0.000,B 0.000,C 90.000,E1 97.530} C_DIS
LIN {X 0.076,Y -464.866,Z 1120.536,A 0.000,B 0.000,C 90.000,E1 96.486} C_DIS
LIN {X 0.208,Y -454.096,Z 1120.528,A 0.000,B 0.000,C 90.000,E1 94.935} C_DIS
LIN {X 0.111,Y -440.052,Z 1120.516,A 0.000,B 0.000,C 90.000,E1 92.865} C_DIS
LIN {X 0.090,Y -427.013,Z 1120.504,A 0.000,B 0.000,C 90.000,E1 90.745} C_DIS
LIN {X -0.130,Y -413.198,Z 1120.491,A 0.000,B 0.000,C 90.000,E1 88.339} C_DIS
LIN {X -0.037,Y -404.288,Z 1120.481,A 0.000,B 0.000,C 90.000,E1 86.674} C_DIS
LIN {X -0.068,Y -393.747,Z 1120.471,A 0.000,B 0.000,C 90.000,E1 84.723} C_DIS
LIN {X 0.138,Y -383.244,Z 1120.460,A 0.000,B 0.000,C 90.000,E1 82.704} C_DIS
LIN {X 0.160,Y -374.209,Z 1120.450,A 0.000,B 0.000,C 90.000,E1 80.971} C_DIS
LIN {X 0.150,Y -366.408,Z 1120.442,A 0.000,B 0.000,C 90.000,E1 79.511} C_DIS
LIN {X -0.002,Y -356.736,Z 1120.432,A 0.000,B 0.000,C 90.000,E1 77.757} C_DIS
LIN {X 0.021,Y -345.180,Z 1120.420,A 0.000,B 0.000,C 90.000,E1 75.644} C_DIS
LIN {X -0.039,Y -333.703,Z 1120.408,A 0.000,B 0.000,C 90.000,E1 73.504} C_DIS
LIN {X -0.095,Y -317.877,Z 1120.391,A 0.000,B 0.000,C 90.000,E1 70.369} C_DIS
LIN {X 0.101,Y -303.145,Z 1120.373,A 0.000,B 0.000,C 90.000,E1 67.102} C_DIS
LIN {X -0.053,Y -290.603,Z 1120.356,A 0.000,B 0.000,C 90.000,E1 64.152} C_DIS
LIN {X 0.003,Y -279.796,Z 1120.341,A 0.000,B 0.000,C 90.000,E1 61.435} C_DIS
LIN {X 0.123,Y -270.657,Z 1120.328,A 0.000,B 0.000,C 90.000,E1 58.997} C_DIS
LIN {X -0.054,Y -258.026,Z 1120.308,A 0.000,B 0.000,C 90.000,E1 55.515} C_DIS
LIN {X -0.035,Y -247.378,Z 1120.290,A 0.000,B 0.000,C 90.000,E1 52.271} C_DIS
LIN {X 0.106,Y -238.478,Z 1120.274,A 0.000,B 0.000,C 90.000,E1 49.299} C_DIS
LIN {X 0.012,Y -230.296,Z 1120.257,A 0.000,B 0.000,C 90.000,E1 46.338} C_DIS
LIN {X 0.032,Y -222.531,Z 1120.241,A 0.000,B 0.000,C 90.000,E1 43.299} C_DIS
LIN {X 0.026,Y -215.055,Z 1120.224,A 0.000,B 0.000,C 90.000,E1 40.216} C_DIS
LIN {X 0.054,Y -207.987,Z 1120.206,A 0.000,B 0.000,C 90.000,E1 37.076} C_DIS
LIN {X -0.005,Y -201.443,Z 1120.188,A 0.000,B 0.000,C 90.000,E1 33.913} C_DIS
LIN {X 0.058,Y -195.448,Z 1120.171,A 0.000,B 0.000,C 90.000,E1 30.669} C_DIS
LIN {X 0.110,Y -190.038,Z 1120.152,A 0.000,B 0.000,C 90.000,E1 27.385} C_DIS
LIN {X -0.065,Y -185.265,Z 1120.134,A 0.000,B 0.000,C 90.000,E1 24.131} C_DIS
LIN {X -0.070,Y -181.142,Z 1120.115,A 0.000,B 0.000,C 90.000,E1 20.791} C_DIS
LIN {X -0.010,Y -176.963,Z 1120.092,A 0.000,B 0.000,C 90.000,E1 16.551} C_DIS
LIN {X -0.034,Y -173.771,Z 1120.068,A 0.000,B 0.000,C 90.000,E1 12.299} C_DIS
LIN {X 0.037,Y -171.360,Z 1120.040,A 0.000,B 0.000,C 90.000,E1 7.125} C_DIS
LIN {X -0.058,Y -172.285,Z 1119.959,A 0.000,B 0.000,C 90.000,E1 352.648} C_DIS
LIN {X 0.035,Y -175.300,Z 1119.930,A 0.000,B 0.000,C 90.000,E1 347.465} C_DIS
LIN {X 0.053,Y -178.885,Z 1119.907,A 0.000,B 0.000,C 90.000,E1 343.196} C_DIS
LIN {X 0.040,Y -183.312,Z 1119.883,A 0.000,B 0.000,C 90.000,E1 338.975} C_DIS
LIN {X 0.081,Y -187.574,Z 1119.865,A 0.000,B 0.000,C 90.000,E1 335.613} C_DIS
LIN {X 0.046,Y -192.548,Z 1119.846,A 0.000,B 0.000,C 90.000,E1 332.308} C_DIS
LIN {X -0.113,Y -198.170,Z 1119.828,A 0.000,B 0.000,C 90.000,E1 329.076} C_DIS
LIN {X 0.014,Y -204.513,Z 1119.810,A 0.000,B 0.000,C 90.000,E1 325.801} C_DIS
LIN {X -0.090,Y -211.655,Z 1119.792,A 0.000,B 0.000,C 90.000,E1 322.637} C_DIS
LIN {X 0.043,Y -219.561,Z 1119.775,A 0.000,B 0.000,C 90.000,E1 319.461} C_DIS
LIN {X 0.048,Y -228.396,Z 1119.758,A 0.000,B 0.000,C 90.000,E1 316.377} C_DIS
LIN {X -0.062,Y -238.201,Z 1119.741,A 0.000,B 0.000,C 90.000,E1 313.380} C_DIS
LIN {X 0.105,Y -249.334,Z 1119.724,A 0.000,B 0.000,C 90.000,E1 310.378} C_DIS
LIN {X 0.007,Y -258.677,Z 1119.712,A 0.000,B 0.000,C 90.000,E1 308.222} C_DIS
LIN {X 0.035,Y -274.320,Z 1119.695,A 0.000,B 0.000,C 90.000,E1 305.025} C_DIS
LIN {X 0.048,Y -291.133,Z 1119.677,A 0.000,B 0.000,C 90.000,E1 301.926} C_DIS
LIN {X -0.092,Y -307.736,Z 1119.663,A 0.000,B 0.000,C 90.000,E1 299.283} C_DIS
LIN {X -0.011,Y -328.118,Z 1119.646,A 0.000,B 0.000,C 90.000,E1 296.360} C_DIS
LIN {X 0.074,Y -345.643,Z 1119.634,A 0.000,B 0.000,C 90.000,E1 294.155} C_DIS
LIN {X 0.002,Y -358.925,Z 1119.626,A 0.000,B 0.000,C 90.000,E1 292.695} C_DIS
LIN {X 0.022,Y -375.034,Z 1119.617,A 0.000,B 0.000,C 90.000,E1 291.099} C_DIS
LIN {X -0.230,Y -394.292,Z 1119.608,A 0.000,B 0.000,C 90.000,E1 289.396} C_DIS
LIN {X -0.149,Y -405.156,Z 1119.602,A 0.000,B 0.000,C 90.000,E1 288.417} C_DIS
LIN {X 0.152,Y -415.672,Z 1119.597,A 0.000,B 0.000,C 90.000,E1 287.402} C_DIS
LIN {X -0.044,Y -423.437,Z 1119.593,A 0.000,B 0.000,C 90.000,E1 286.677} C_DIS
LIN {X 0.082,Y -430.938,Z 1119.588,A 0.000,B 0.000,C 90.000,E1 285.898} C_DIS
LIN {X -0.148,Y -438.243,Z 1119.584,A 0.000,B 0.000,C 90.000,E1 285.134} C_DIS
LIN {X 0.145,Y -445.052,Z 1119.580,A 0.000,B 0.000,C 90.000,E1 284.300} C_DIS
LIN {X -0.034,Y -451.313,Z 1119.575,A 0.000,B 0.000,C 90.000,E1 283.536} C_DIS
LIN {X -0.167,Y -456.841,Z 1119.571,A 0.000,B 0.000,C 90.000,E1 282.771} C_DIS
LIN {X -0.247,Y -461.633,Z 1119.567,A 0.000,B 0.000,C 90.000,E1 282.007} C_DIS
LIN {X 0.165,Y -465.807,Z 1119.562,A 0.000,B 0.000,C 90.000,E1 281.186} C_DIS
LIN {X 0.075,Y -469.440,Z 1119.558,A 0.000,B 0.000,C 90.000,E1 280.433} C_DIS
LIN {X 0.097,Y -472.470,Z 1119.554,A 0.000,B 0.000,C 90.000,E1 279.670} C_DIS
LIN {X 0.198,Y -474.170,Z 1119.551,A 0.000,B 0.000,C 90.000,E1 279.151} C_DIS
LIN {X -0.085,Y -475.594,Z 1119.548,A 0.000,B 0.000,C 90.000,E1 278.681} C_DIS
LIN {X 0.039,Y -476.744,Z 1119.545,A 0.000,B 0.000,C 90.000,E1 278.163} C_DIS
LIN {X 0.174,Y -477.617,Z 1119.543,A 0.000,B 0.000,C 90.000,E1 277.644} C_DIS
LIN {X -0.158,Y -478.193,Z 1119.540,A 0.000,B 0.000,C 90.000,E1 277.182} C_DIS
LIN {X -0.009,Y -478.422,Z 1119.537,A 0.000,B 0.000,C 90.000,E1 276.663} C_DIS
LIN {X 0.145,Y -478.401,Z 1119.534,A 0.000,B 0.000,C 90.000,E1 276.144} C_DIS
LIN {X -0.178,Y -478.000,Z 1119.531,A 0.000,B 0.000,C 90.000,E1 275.682} C_DIS
LIN {X -0.026,Y -477.336,Z 1119.529,A 0.000,B 0.000,C 90.000,E1 275.163} C_DIS
LIN {X 0.122,Y -476.247,Z 1119.526,A 0.000,B 0.000,C 90.000,E1 274.645} C_DIS
LIN {X -0.246,Y -474.746,Z 1119.523,A 0.000,B 0.000,C 90.000,E1 274.188} C_DIS
LIN {X -0.108,Y -472.713,Z 1119.520,A 0.000,B 0.000,C 90.000,E1 273.669} C_DIS
LIN {X -0.011,Y -470.020,Z 1119.517,A 0.000,B 0.000,C 90.000,E1 273.154} C_DIS
LIN {X 0.092,Y -466.499,Z 1119.515,A 0.000,B 0.000,C 90.000,E1 272.636} C_DIS
LIN {X 0.155,Y -461.892,Z 1119.512,A 0.000,B 0.000,C 90.000,E1 272.121} C_DIS
LIN {X -0.055,Y -459.102,Z 1119.510,A 0.000,B 0.000,C 90.000,E1 271.892} C_DIS
LIN {X -0.152,Y -452.977,Z 1119.508,A 0.000,B 0.000,C 90.000,E1 271.432} C_DIS
LIN {X -0.118,Y -446.344,Z 1119.506,A 0.000,B 0.000,C 90.000,E1 271.031} C_DIS
LIN {X -0.021,Y -439.460,Z 1119.504,A 0.000,B 0.000,C 90.000,E1 270.688} C_DIS
LIN {X 0.050,Y -432.440,Z 1119.502,A 0.000,B 0.000,C 90.000,E1 270.401} C_DIS
LIN {X 0.034,Y -425.342,Z 1119.501,A 0.000,B 0.000,C 90.000,E1 270.172} C_DIS
LIN {X -0.124,Y -418.261,Z 1119.500,A 0.000,B 0.000,C 90.000,E1 270.000} C_DIS
LIN {X -0.012,Y -410.833,Z 1119.499,A 0.000,B 0.000,C 90.000,E1 269.828} C_DIS
LIN {X -0.088,Y -403.017,Z 1119.498,A 0.000,B 0.000,C 90.000,E1 269.714} C_DIS
LIN {X 0.015,Y -392.546,Z 1119.498,A 0.000,B 0.000,C 90.000,E1 269.599} C_DIS
LIN {X 0.180,Y -383.723,Z 1119.498,A 0.000,B 0.000,C 90.000,E1 269.542} C_DIS
LIN {X 0.051,Y -181.453,Z 1119.498,A 0.000,B 0.000,C 90.000,E1 269.542} C_DIS
LIN {X -0.007,Y -180.863,Z 1119.472,A 0.000,B 0.000,C 90.000,E1 265.008} C_DIS
LIN {X 0.046,Y -178.976,Z 1119.444,A 0.000,B 0.000,C 90.000,E1 259.926} C_DIS
LIN {X 0.056,Y -177.942,Z 1119.435,A 0.000,B 0.000,C 90.000,E1 258.229} C_DIS
LIN {X 0.071,Y -175.582,Z 1119.411,A 0.000,B 0.000,C 90.000,E1 253.976} C_DIS
LIN {X 0.077,Y -172.308,Z 1119.387,A 0.000,B 0.000,C 90.000,E1 249.699} C_DIS
LIN {X 0.055,Y -171.787,Z 1119.383,A 0.000,B 0.000,C 90.000,E1 248.847} C_DIS
LIN {X -0.068,Y -169.454,Z 1119.368,A 0.000,B 0.000,C 90.000,E1 246.305} C_DIS
LIN {X -0.012,Y -166.783,Z 1119.349,A 0.000,B 0.000,C 90.000,E1 242.820} C_DIS
LIN {X -0.016,Y -162.763,Z 1119.325,A 0.000,B 0.000,C 90.000,E1 238.456} C_DIS
LIN {X -0.040,Y -161.453,Z 1119.315,A 0.000,B 0.000,C 90.000,E1 236.707} C_DIS
LIN {X 0.002,Y -157.447,Z 1119.290,A 0.000,B 0.000,C 90.000,E1 232.271} C_DIS
LIN {X -0.065,Y -155.456,Z 1119.276,A 0.000,B 0.000,C 90.000,E1 229.622} C_DIS
LIN {X 0.084,Y -151.772,Z 1119.251,A 0.000,B 0.000,C 90.000,E1 225.081} C_DIS
LIN {X -0.006,Y -149.976,Z 1119.236,A 0.000,B 0.000,C 90.000,E1 222.405} C_DIS
LIN {X 0.005,Y -146.812,Z 1119.210,A 0.000,B 0.000,C 90.000,E1 217.855} C_DIS
LIN {X 0.022,Y -145.389,Z 1119.195,A 0.000,B 0.000,C 90.000,E1 215.105} C_DIS
LIN {X -0.060,Y -142.826,Z 1119.170,A 0.000,B 0.000,C 90.000,E1 210.541} C_DIS
LIN {X -0.004,Y -141.439,Z 1119.149,A 0.000,B 0.000,C 90.000,E1 206.821} C_DIS
LIN {X 0.041,Y -139.368,Z 1119.113,A 0.000,B 0.000,C 90.000,E1 200.301} C_DIS
LIN {X 0.027,Y -138.815,Z 1119.097,A 0.000,B 0.000,C 90.000,E1 197.511} C_DIS
LIN {X -0.059,Y -138.352,Z 1119.056,A 0.000,B 0.000,C 90.000,E1 190.074} C_DIS
LIN {X 0.054,Y -139.538,Z 1119.004,A 0.000,B 0.000,C 90.000,E1 180.688} C_DIS
LIN {X 0.006,Y -141.229,Z 1118.973,A 0.000,B 0.000,C 90.000,E1 175.122} C_DIS
LIN {X -0.035,Y -142.601,Z 1118.957,A 0.000,B 0.000,C 90.000,E1 172.356} C_DIS
LIN {X 0.059,Y -144.907,Z 1118.932,A 0.000,B 0.000,C 90.000,E1 167.701} C_DIS
LIN {X 0.012,Y -147.536,Z 1118.911,A 0.000,B 0.000,C 90.000,E1 164.047} C_DIS
LIN {X -0.056,Y -150.135,Z 1118.891,A 0.000,B 0.000,C 90.000,E1 160.423} C_DIS
LIN {X -0.045,Y -153.501,Z 1118.871,A 0.000,B 0.000,C 90.000,E1 156.794} C_DIS
LIN {X 0.018,Y -157.866,Z 1118.846,A 0.000,B 0.000,C 90.000,E1 152.281} C_DIS
LIN {X -0.027,Y -162.152,Z 1118.826,A 0.000,B 0.000,C 90.000,E1 148.742} C_DIS
LIN {X 0.088,Y -166.357,Z 1118.807,A 0.000,B 0.000,C 90.000,E1 145.182} C_DIS
LIN {X -0.043,Y -171.375,Z 1118.787,A 0.000,B 0.000,C 90.000,E1 141.743} C_DIS
LIN {X 0.000,Y -176.283,Z 1118.768,A 0.000,B 0.000,C 90.000,E1 138.286} C_DIS
LIN {X 0.002,Y -180.568,Z 1118.754,A 0.000,B 0.000,C 90.000,E1 135.729} C_DIS
LIN {X -0.020,Y -185.970,Z 1118.735,A 0.000,B 0.000,C 90.000,E1 132.366} C_DIS
LIN {X 0.035,Y -190.602,Z 1118.721,A 0.000,B 0.000,C 90.000,E1 129.850} C_DIS
LIN {X -0.057,Y -196.353,Z 1118.703,A 0.000,B 0.000,C 90.000,E1 126.583} C_DIS
LIN {X -0.002,Y -200.564,Z 1118.691,A 0.000,B 0.000,C 90.000,E1 124.452} C_DIS
LIN {X -0.056,Y -308.924,Z 1118.691,A 0.000,B 0.000,C 90.000,E1 124.452} C_DIS
LIN {X 0.092,Y -310.306,Z 1118.691,A 0.000,B 0.000,C 90.000,E1 124.405} C_DIS
LIN {X 0.032,Y -316.311,Z 1118.690,A 0.000,B 0.000,C 90.000,E1 124.119} C_DIS
LIN {X -0.080,Y -319.376,Z 1118.688,A 0.000,B 0.000,C 90.000,E1 123.833} C_DIS
LIN {X 0.084,Y -322.985,Z 1118.685,A 0.000,B 0.000,C 90.000,E1 123.245} C_DIS
LIN {X -0.107,Y -324.425,Z 1118.683,A 0.000,B 0.000,C 90.000,E1 122.959} C_DIS
LIN {X -0.035,Y -336.291,Z 1118.666,A 0.000,B 0.000,C 90.000,E1 119.795} C_DIS
LIN {X 0.050,Y -348.368,Z 1118.650,A 0.000,B 0.000,C 90.000,E1 117.001} C_DIS
LIN {X 0.028,Y -361.915,Z 1118.635,A 0.000,B 0.000,C 90.000,E1 114.283} C_DIS
LIN {X 0.141,Y -375.291,Z 1118.622,A 0.000,B 0.000,C 90.000,E1 111.897} C_DIS
LIN {X 0.170,Y -390.021,Z 1118.609,A 0.000,B 0.000,C 90.000,E1 109.577} C_DIS
LIN {X 0.061,Y -406.205,Z 1118.596,A 0.000,B 0.000,C 90.000,E1 107.330} C_DIS
LIN {X -0.018,Y -423.962,Z 1118.584,A 0.000,B 0.000,C 90.000,E1 105.134} C_DIS
LIN {X -0.110,Y -443.329,Z 1118.572,A 0.000,B 0.000,C 90.000,E1 103.008} C_DIS
LIN {X -0.001,Y -463.531,Z 1118.561,A 0.000,B 0.000,C 90.000,E1 101.007} C_DIS
LIN {X -0.081,Y -468.618,Z 1118.558,A 0.000,B 0.000,C 90.000,E1 100.546} C_DIS
LIN {X -0.058,Y -470.611,Z 1118.557,A 0.000,B 0.000,C 90.000,E1 100.310} C_DIS
LIN {X 0.258,Y -472.249,Z 1118.556,A 0.000,B 0.000,C 90.000,E1 100.018} C_DIS
LIN {X 0.029,Y -473.477,Z 1118.554,A 0.000,B 0.000,C 90.000,E1 99.792} C_DIS
LIN {X 0.218,Y -474.982,Z 1118.552,A 0.000,B 0.000,C 90.000,E1 99.265} C_DIS
LIN {X -0.132,Y -475.445,Z 1118.549,A 0.000,B 0.000,C 90.000,E1 98.803} C_DIS
LIN {X 0.067,Y -474.945,Z 1118.546,A 0.000,B 0.000,C 90.000,E1 98.276} C_DIS
LIN {X 0.199,Y -473.405,Z 1118.543,A 0.000,B 0.000,C 90.000,E1 97.757} C_DIS
LIN {X -0.002,Y -472.165,Z 1118.542,A 0.000,B 0.000,C 90.000,E1 97.530} C_DIS
LIN {X 0.122,Y -468.649,Z 1118.539,A 0.000,B 0.000,C 90.000,E1 97.011} C_DIS
LIN {X 0.189,Y -456.041,Z 1118.529,A 0.000,B 0.000,C 90.000,E1 95.220} C_DIS
LIN {X -0.130,Y -440.176,Z 1118.516,A 0.000,B 0.000,C 90.000,E1 92.922} C_DIS
LIN {X -0.141,Y -427.134,Z 1118.504,A 0.000,B 0.000,C 90.000,E1 90.802} C_DIS
LIN {X 0.061,Y -413.322,Z 1118.491,A 0.000,B 0.000,C 90.000,E1 88.339} C_DIS
LIN {X 0.153,Y -404.390,Z 1118.482,A 0.000,B 0.000,C 90.000,E1 86.674} C_DIS
LIN {X 0.119,Y -393.848,Z 1118.471,A 0.000,B 0.000,C 90.000,E1 84.723} C_DIS
LIN {X -0.058,Y -383.320,Z 1118.460,A 0.000,B 0.000,C 90.000,E1 82.761} C_DIS
LIN {X -0.029,Y -374.278,Z 1118.450,A 0.000,B 0.000,C 90.000,E1 81.027} C_DIS
LIN {X -0.031,Y -366.497,Z 1118.442,A 0.000,B 0.000,C 90.000,E1 79.567} C_DIS
LIN {X 0.174,Y -356.791,Z 1118.432,A 0.000,B 0.000,C 90.000,E1 77.757} C_DIS
LIN {X -0.142,Y -345.254,Z 1118.420,A 0.000,B 0.000,C 90.000,E1 75.700} C_DIS
LIN {X 0.110,Y -332.140,Z 1118.407,A 0.000,B 0.000,C 90.000,E1 73.196} C_DIS
LIN {X 0.008,Y -316.412,Z 1118.389,A 0.000,B 0.000,C 90.000,E1 70.061} C_DIS
LIN {X 0.155,Y -301.759,Z 1118.371,A 0.000,B 0.000,C 90.000,E1 66.794} C_DIS
LIN {X -0.046,Y -289.268,Z 1118.355,A 0.000,B 0.000,C 90.000,E1 63.845} C_DIS
LIN {X -0.030,Y -278.502,Z 1118.340,A 0.000,B 0.000,C 90.000,E1 61.129} C_DIS
LIN {X -0.173,Y -269.369,Z 1118.326,A 0.000,B 0.000,C 90.000,E1 58.742} C_DIS
LIN {X 0.080,Y -258.008,Z 1118.308,A 0.000,B 0.000,C 90.000,E1 55.515} C_DIS
LIN {X 0.101,Y -246.193,Z 1118.288,A 0.000,B 0.000,C 90.000,E1 51.904} C_DIS
LIN {X 0.014,Y -236.291,Z 1118.270,A 0.000,B 0.000,C 90.000,E1 48.609} C_DIS
LIN {X -0.130,Y -228.187,Z 1118.253,A 0.000,B 0.000,C 90.000,E1 45.648} C_DIS
LIN {X 0.006,Y -220.474,Z 1118.236,A 0.000,B 0.000,C 90.000,E1 42.567} C_DIS
LIN {X -0.041,Y -213.065,Z 1118.219,A 0.000,B 0.000,C 90.000,E1 39.483} C_DIS
LIN {X 0.104,Y -206.120,Z 1118.202,A 0.000,B 0.000,C 90.000,E1 36.297} C_DIS
LIN {X -0.112,Y -199.667,Z 1118.184,A 0.000,B 0.000,C 90.000,E1 33.166} C_DIS
LIN {X 0.077,Y -193.820,Z 1118.166,A 0.000,B 0.000,C 90.000,E1 29.873} C_DIS
LIN {X 0.000,Y -188.544,Z 1118.148,A 0.000,B 0.000,C 90.000,E1 26.616} C_DIS
LIN {X -0.115,Y -183.930,Z 1118.129,A 0.000,B 0.000,C 90.000,E1 23.334} C_DIS
LIN {X 0.021,Y -179.973,Z 1118.111,A 0.000,B 0.000,C 90.000,E1 19.939} C_DIS
LIN {X -0.011,Y -175.984,Z 1118.087,A 0.000,B 0.000,C 90.000,E1 15.717} C_DIS
LIN {X 0.066,Y -172.996,Z 1118.064,A 0.000,B 0.000,C 90.000,E1 11.422} C_DIS
LIN {X -0.076,Y -170.613,Z 1118.030,A 0.000,B 0.000,C 90.000,E1 5.448} C_DIS
LIN {X -0.086,Y -171.632,Z 1117.964,A 0.000,B 0.000,C 90.000,E1 353.514} C_DIS
LIN {X -0.050,Y -174.379,Z 1117.935,A 0.000,B 0.000,C 90.000,E1 348.342} C_DIS
LIN {X 0.018,Y -177.791,Z 1117.911,A 0.000,B 0.000,C 90.000,E1 344.047} C_DIS
LIN {X -0.035,Y -182.015,Z 1117.888,A 0.000,B 0.000,C 90.000,E1 339.826} C_DIS
LIN {X -0.096,Y -186.114,Z 1117.869,A 0.000,B 0.000,C 90.000,E1 336.485} C_DIS
LIN {X 0.004,Y -190.942,Z 1117.851,A 0.000,B 0.000,C 90.000,E1 333.127} C_DIS
LIN {X -0.116,Y -196.433,Z 1117.832,A 0.000,B 0.000,C 90.000,E1 329.871} C_DIS
LIN {X 0.027,Y -202.580,Z 1117.814,A 0.000,B 0.000,C 90.000,E1 326.580} C_DIS
LIN {X -0.127,Y -209.571,Z 1117.797,A 0.000,B 0.000,C 90.000,E1 323.417} C_DIS
LIN {X -0.024,Y -217.288,Z 1117.779,A 0.000,B 0.000,C 90.000,E1 320.231} C_DIS
LIN {X -0.083,Y -225.885,Z 1117.762,A 0.000,B 0.000,C 90.000,E1 317.148} C_DIS
LIN {X -0.092,Y -235.473,Z 1117.745,A 0.000,B 0.000,C 90.000,E1 314.109} C_DIS
LIN {X 0.005,Y -246.288,Z 1117.728,A 0.000,B 0.000,C 90.000,E1 311.105} C_DIS
LIN {X 0.018,Y -255.363,Z 1117.716,A 0.000,B 0.000,C 90.000,E1 308.910} C_DIS
LIN {X 0.037,Y -263.655,Z 1117.706,A 0.000,B 0.000,C 90.000,E1 307.111} C_DIS
LIN {X -0.033,Y -276.109,Z 1117.693,A 0.000,B 0.000,C 90.000,E1 304.659} C_DIS
LIN {X 0.121,Y -293.180,Z 1117.675,A 0.000,B 0.000,C 90.000,E1 301.544} C_DIS
LIN {X 0.161,Y -307.808,Z 1117.662,A 0.000,B 0.000,C 90.000,E1 299.205} C_DIS
LIN {X -0.187,Y -328.222,Z 1117.646,A 0.000,B 0.000,C 90.000,E1 296.360} C_DIS
LIN {X 0.035,Y -345.781,Z 1117.634,A 0.000,B 0.000,C 90.000,E1 294.131} C_DIS
LIN {X 0.181,Y -359.025,Z 1117.626,A 0.000,B 0.000,C 90.000,E1 292.642} C_DIS
LIN {X 0.128,Y -372.761,Z 1117.618,A 0.000,B 0.000,C 90.000,E1 291.280} C_DIS
LIN {X 0.067,Y -394.512,Z 1117.607,A 0.000,B 0.000,C 90.000,E1 289.322} C_DIS
LIN {X 0.024,Y -405.352,Z 1117.602,A 0.000,B 0.000,C 90.000,E1 288.362} C_DIS
LIN {X -0.046,Y -415.865,Z 1117.597,A 0.000,B 0.000,C 90.000,E1 287.402} C_DIS
LIN {X 0.068,Y -426.197,Z 1117.591,A 0.000,B 0.000,C 90.000,E1 286.386} C_DIS
LIN {X 0.134,Y -433.612,Z 1117.587,A 0.000,B 0.000,C 90.000,E1 285.607} C_DIS
LIN {X 0.014,Y -440.741,Z 1117.582,A 0.000,B 0.000,C 90.000,E1 284.828} C_DIS
LIN {X -0.207,Y -447.431,Z 1117.578,A 0.000,B 0.000,C 90.000,E1 284.064} C_DIS
LIN {X 0.065,Y -453.466,Z 1117.574,A 0.000,B 0.000,C 90.000,E1 283.244} C_DIS
LIN {X -0.041,Y -458.751,Z 1117.569,A 0.000,B 0.000,C 90.000,E1 282.479} C_DIS
LIN {X -0.108,Y -463.362,Z 1117.565,A 0.000,B 0.000,C 90.000,E1 281.715} C_DIS
LIN {X -0.133,Y -467.339,Z 1117.561,A 0.000,B 0.000,C 90.000,E1 280.950} C_DIS
LIN {X -0.217,Y -470.746,Z 1117.557,A 0.000,B 0.000,C 90.000,E1 280.197} C_DIS
LIN {X -0.043,Y -472.702,Z 1117.554,A 0.000,B 0.000,C 90.000,E1 279.670} C_DIS
LIN {X 0.058,Y -474.425,Z 1117.551,A 0.000,B 0.000,C 90.000,E1 279.151} C_DIS
LIN {X 0.247,Y -475.823,Z 1117.548,A 0.000,B 0.000,C 90.000,E1 278.624} C_DIS
LIN {X -0.098,Y -476.984,Z 1117.545,A 0.000,B 0.000,C 90.000,E1 278.163} C_DIS
LIN {X 0.038,Y -477.835,Z 1117.542,A 0.000,B 0.000,C 90.000,E1 277.644} C_DIS
LIN {X 0.183,Y -478.395,Z 1117.540,A 0.000,B 0.000,C 90.000,E1 277.125} C_DIS
LIN {X -0.142,Y -478.703,Z 1117.537,A 0.000,B 0.000,C 90.000,E1 276.663} C_DIS
LIN {X 0.012,Y -478.649,Z 1117.534,A 0.000,B 0.000,C 90.000,E1 276.144} C_DIS
LIN {X 0.167,Y -478.284,Z 1117.531,A 0.000,B 0.000,C 90.000,E1 275.625} C_DIS
LIN {X -0.155,Y -477.589,Z 1117.529,A 0.000,B 0.000,C 90.000,E1 275.163} C_DIS
LIN {X -0.005,Y -476.544,Z 1117.526,A 0.000,B 0.000,C 90.000,E1 274.645} C_DIS
LIN {X 0.103,Y -475.017,Z 1117.523,A 0.000,B 0.000,C 90.000,E1 274.131} C_DIS
LIN {X -0.232,Y -472.979,Z 1117.520,A 0.000,B 0.000,C 90.000,E1 273.669} C_DIS
LIN {X -0.106,Y -470.305,Z 1117.517,A 0.000,B 0.000,C 90.000,E1 273.151} C_DIS
LIN {X -0.026,Y -466.805,Z 1117.515,A 0.000,B 0.000,C 90.000,E1 272.636} C_DIS
LIN {X 0.039,Y -462.201,Z 1117.512,A 0.000,B 0.000,C 90.000,E1 272.121} C_DIS
LIN {X -0.169,Y -459.420,Z 1117.510,A 0.000,B 0.000,C 90.000,E1 271.892} C_DIS
LIN {X 0.175,Y -453.323,Z 1117.508,A 0.000,B 0.000,C 90.000,E1 271.375} C_DIS
LIN {X -0.194,Y -449.909,Z 1117.507,A 0.000,B 0.000,C 90.000,E1 271.203} C_DIS
LIN {X 0.080,Y -443.070,Z 1117.505,A 0.000,B 0.000,C 90.000,E1 270.802} C_DIS
LIN {X -0.054,Y -436.051,Z 1117.503,A 0.000,B 0.000,C 90.000,E1 270.516} C_DIS
LIN {X 0.212,Y -428.986,Z 1117.501,A 0.000,B 0.000,C 90.000,E1 270.229} C_DIS
LIN {X 0.134,Y -418.497,Z 1117.500,A 0.000,B 0.000,C 90.000,E1 269.943} C_DIS
LIN {X -0.180,Y -411.022,Z 1117.499,A 0.000,B 0.000,C 90.000,E1 269.828} C_DIS
LIN {X 0.141,Y -402.874,Z 1117.498,A 0.000,B 0.000,C 90.000,E1 269.656} C_DIS
LIN {X -0.141,Y -391.705,Z 1117.498,A 0.000,B 0.000,C 90.000,E1 269.599} C_DIS
LIN {X 0.105,Y -386.736,Z 1117.498,A 0.000,B 0.000,C 90.000,E1 269.542} C_DIS
LIN {X 0.016,Y -181.451,Z 1117.497,A 0.000,B 0.000,C 90.000,E1 269.542} C_DIS
LIN {X -0.042,Y -180.861,Z 1117.472,A 0.000,B 0.000,C 90.000,E1 265.008} C_DIS
LIN {X 0.011,Y -178.974,Z 1117.444,A 0.000,B 0.000,C 90.000,E1 259.926} C_DIS
LIN {X 0.022,Y -177.934,Z 1117.435,A 0.000,B 0.000,C 90.000,E1 258.229} C_DIS
LIN {X 0.036,Y -175.574,Z 1117.411,A 0.000,B 0.000,C 90.000,E1 253.976} C_DIS
LIN {X 0.043,Y -172.301,Z 1117.387,A 0.000,B 0.000,C 90.000,E1 249.699} C_DIS
LIN {X 0.021,Y -171.780,Z 1117.383,A 0.000,B 0.000,C 90.000,E1 248.847} C_DIS
LIN {X -0.007,Y -168.710,Z 1117.363,A 0.000,B 0.000,C 90.000,E1 245.409} C_DIS
LIN {X 0.031,Y -166.774,Z 1117.349,A 0.000,B 0.000,C 90.000,E1 242.794} C_DIS
LIN {X -0.049,Y -162.754,Z 1117.325,A 0.000,B 0.000,C 90.000,E1 238.456} C_DIS
LIN {X -0.073,Y -161.444,Z 1117.315,A 0.000,B 0.000,C 90.000,E1 236.707} C_DIS
LIN {X -0.031,Y -157.437,Z 1117.290,A 0.000,B 0.000,C 90.000,E1 232.271} C_DIS
LIN {X 0.004,Y -155.445,Z 1117.276,A 0.000,B 0.000,C 90.000,E1 229.585} C_DIS
LIN {X 0.053,Y -151.764,Z 1117.251,A 0.000,B 0.000,C 90.000,E1 225.081} C_DIS
LIN {X 0.064,Y -149.966,Z 1117.235,A 0.000,B 0.000,C 90.000,E1 222.366} C_DIS
LIN {X -0.025,Y -146.805,Z 1117.210,A 0.000,B 0.000,C 90.000,E1 217.855} C_DIS
LIN {X -0.010,Y -145.382,Z 1117.195,A 0.000,B 0.000,C 90.000,E1 215.105} C_DIS
LIN {X -0.018,Y -142.442,Z 1117.164,A 0.000,B 0.000,C 90.000,E1 209.589} C_DIS
LIN {X 0.029,Y -141.433,Z 1117.149,A 0.000,B 0.000,C 90.000,E1 206.796} C_DIS
LIN {X 0.011,Y -139.366,Z 1117.113,A 0.000,B 0.000,C 90.000,E1 200.301} C_DIS
LIN {X -0.004,Y -138.812,Z 1117.097,A 0.000,B 0.000,C 90.000,E1 197.511} C_DIS
LIN {X 0.048,Y -138.351,Z 1117.056,A 0.000,B 0.000,C 90.000,E1 190.018} C_DIS
LIN {X 0.024,Y -139.540,Z 1117.004,A 0.000,B 0.000,C 90.000,E1 180.688} C_DIS
LIN {X -0.024,Y -141.235,Z 1116.973,A 0.000,B 0.000,C 90.000,E1 175.122} C_DIS
LIN {X -0.066,Y -142.605,Z 1116.957,A 0.000,B 0.000,C 90.000,E1 172.356} C_DIS
LIN {X 0.029,Y -144.915,Z 1116.932,A 0.000,B 0.000,C 90.000,E1 167.701} C_DIS
LIN {X 0.022,Y -147.544,Z 1116.911,A 0.000,B 0.000,C 90.000,E1 164.031} C_DIS
LIN {X 0.054,Y -150.145,Z 1116.891,A 0.000,B 0.000,C 90.000,E1 160.369} C_DIS
LIN {X 0.064,Y -153.514,Z 1116.871,A 0.000,B 0.000,C 90.000,E1 156.741} C_DIS
LIN {X -0.015,Y -157.879,Z 1116.846,A 0.000,B 0.000,C 90.000,E1 152.281} C_DIS
LIN {X -0.060,Y -162.165,Z 1116.826,A 0.000,B 0.000,C 90.000,E1 148.742} C_DIS
LIN {X 0.055,Y -166.373,Z 1116.807,A 0.000,B 0.000,C 90.000,E1 145.182} C_DIS
LIN {X 0.057,Y -171.389,Z 1116.787,A 0.000,B 0.000,C 90.000,E1 141.698} C_DIS
LIN {X 0.097,Y -176.301,Z 1116.768,A 0.000,B 0.000,C 90.000,E1 138.243} C_DIS
LIN {X -0.034,Y -180.587,Z 1116.754,A 0.000,B 0.000,C 90.000,E1 135.729} C_DIS
LIN {X -0.057,Y -185.989,Z 1116.735,A 0.000,B 0.000,C 90.000,E1 132.366} C_DIS
LIN {X -0.001,Y -190.622,Z 1116.721,A 0.000,B 0.000,C 90.000,E1 129.850} C_DIS
LIN {X -0.095,Y -196.373,Z 1116.703,A 0.000,B 0.000,C 90.000,E1 126.583} C_DIS
LIN {X 0.003,Y -200.497,Z 1116.692,A 0.000,B 0.000,C 90.000,E1 124.485} C_DIS
LIN {X -0.056,Y -308.964,Z 1116.692,A 0.000,B 0.000,C 90.000,E1 124.485} C_DIS
LIN {X -0.001,Y -310.361,Z 1116.691,A 0.000,B 0.000,C 90.000,E1 124.452} C_DIS
LIN {X 0.026,Y -314.420,Z 1116.690,A 0.000,B 0.000,C 90.000,E1 124.278} C_DIS
LIN {X -0.028,Y -316.706,Z 1116.690,A 0.000,B 0.000,C 90.000,E1 124.119} C_DIS
LIN {X 0.098,Y -320.575,Z 1116.687,A 0.000,B 0.000,C 90.000,E1 123.658} C_DIS
LIN {X -0.017,Y -322.451,Z 1116.685,A 0.000,B 0.000,C 90.000,E1 123.372} C_DIS
LIN {X -0.134,Y -323.921,Z 1116.684,A 0.000,B 0.000,C 90.000,E1 123.086} C_DIS
LIN {X 0.056,Y -337.045,Z 1116.664,A 0.000,B 0.000,C 90.000,E1 119.589} C_DIS
LIN {X 0.004,Y -349.219,Z 1116.649,A 0.000,B 0.000,C 90.000,E1 116.821} C_DIS
LIN {X 0.161,Y -362.870,Z 1116.634,A 0.000,B 0.000,C 90.000,E1 114.079} C_DIS
LIN {X 0.153,Y -376.345,Z 1116.621,A 0.000,B 0.000,C 90.000,E1 111.716} C_DIS
LIN {X -0.157,Y -391.181,Z 1116.608,A 0.000,B 0.000,C 90.000,E1 109.450} C_DIS
LIN {X 0.012,Y -407.482,Z 1116.595,A 0.000,B 0.000,C 90.000,E1 107.166} C_DIS
LIN {X 0.088,Y -425.363,Z 1116.583,A 0.000,B 0.000,C 90.000,E1 104.954} C_DIS
LIN {X 0.058,Y -444.832,Z 1116.571,A 0.000,B 0.000,C 90.000,E1 102.827} C_DIS
LIN {X 0.185,Y -465.076,Z 1116.560,A 0.000,B 0.000,C 90.000,E1 100.838} C_DIS
LIN {X 0.182,Y -467.659,Z 1116.559,A 0.000,B 0.000,C 90.000,E1 100.602} C_DIS
LIN {X 0.219,Y -469.874,Z 1116.558,A 0.000,B 0.000,C 90.000,E1 100.366} C_DIS
LIN {X 0.172,Y -471.547,Z 1116.556,A 0.000,B 0.000,C 90.000,E1 100.141} C_DIS
LIN {X 0.028,Y -472.940,Z 1116.555,A 0.000,B 0.000,C 90.000,E1 99.905} C_DIS
LIN {X -0.118,Y -473.976,Z 1116.554,A 0.000,B 0.000,C 90.000,E1 99.670} C_DIS
LIN {X -0.004,Y -475.172,Z 1116.551,A 0.000,B 0.000,C 90.000,E1 99.151} C_DIS
LIN {X 0.191,Y -475.366,Z 1116.548,A 0.000,B 0.000,C 90.000,E1 98.624} C_DIS
LIN {X -0.148,Y -474.590,Z 1116.545,A 0.000,B 0.000,C 90.000,E1 98.163} C_DIS
LIN {X -0.015,Y -472.722,Z 1116.542,A 0.000,B 0.000,C 90.000,E1 97.644} C_DIS
LIN {X -0.154,Y -471.267,Z 1116.541,A 0.000,B 0.000,C 90.000,E1 97.409} C_DIS
LIN {X 0.189,Y -456.796,Z 1116.530,A 0.000,B 0.000,C 90.000,E1 95.334} C_DIS
LIN {X -0.109,Y -440.880,Z 1116.517,A 0.000,B 0.000,C 90.000,E1 93.037} C_DIS
LIN {X -0.106,Y -427.822,Z 1116.505,A 0.000,B 0.000,C 90.000,E1 90.917} C_DIS
LIN {X 0.109,Y -413.947,Z 1116.491,A 0.000,B 0.000,C 90.000,E1 88.453} C_DIS
LIN {X 0.211,Y -405.034,Z 1116.482,A 0.000,B 0.000,C 90.000,E1 86.788} C_DIS
LIN {X 0.195,Y -394.476,Z 1116.471,A 0.000,B 0.000,C 90.000,E1 84.837} C_DIS
LIN {X 0.015,Y -382.438,Z 1116.459,A 0.000,B 0.000,C 90.000,E1 82.591} C_DIS
LIN {X 0.080,Y -373.363,Z 1116.449,A 0.000,B 0.000,C 90.000,E1 80.849} C_DIS
LIN {X -0.001,Y -365.526,Z 1116.441,A 0.000,B 0.000,C 90.000,E1 79.398} C_DIS
LIN {X -0.169,Y -355.785,Z 1116.431,A 0.000,B 0.000,C 90.000,E1 77.645} C_DIS
LIN {X -0.081,Y -344.224,Z 1116.419,A 0.000,B 0.000,C 90.000,E1 75.519} C_DIS
LIN {X 0.050,Y -331.116,Z 1116.406,A 0.000,B 0.000,C 90.000,E1 73.032} C_DIS
LIN {X 0.012,Y -315.477,Z 1116.388,A 0.000,B 0.000,C 90.000,E1 69.880} C_DIS
LIN {X -0.047,Y -302.303,Z 1116.372,A 0.000,B 0.000,C 90.000,E1 66.975} C_DIS
LIN {X -0.080,Y -291.149,Z 1116.357,A 0.000,B 0.000,C 90.000,E1 64.332} C_DIS
LIN {X -0.138,Y -280.316,Z 1116.342,A 0.000,B 0.000,C 90.000,E1 61.641} C_DIS
LIN {X -0.002,Y -271.157,Z 1116.329,A 0.000,B 0.000,C 90.000,E1 59.203} C_DIS
LIN {X 0.055,Y -258.421,Z 1116.309,A 0.000,B 0.000,C 90.000,E1 55.674} C_DIS
LIN {X 0.082,Y -246.545,Z 1116.289,A 0.000,B 0.000,C 90.000,E1 52.065} C_DIS
LIN {X 0.014,Y -237.621,Z 1116.273,A 0.000,B 0.000,C 90.000,E1 49.138} C_DIS
LIN {X 0.070,Y -229.415,Z 1116.256,A 0.000,B 0.000,C 90.000,E1 46.134} C_DIS
LIN {X 0.067,Y -221.625,Z 1116.240,A 0.000,B 0.000,C 90.000,E1 43.095} C_DIS
LIN {X 0.045,Y -214.127,Z 1116.222,A 0.000,B 0.000,C 90.000,E1 40.011} C_DIS
LIN {X 0.052,Y -207.067,Z 1116.205,A 0.000,B 0.000,C 90.000,E1 36.870} C_DIS
LIN {X -0.028,Y -200.508,Z 1116.187,A 0.000,B 0.000,C 90.000,E1 33.706} C_DIS
LIN {X 0.012,Y -194.552,Z 1116.169,A 0.000,B 0.000,C 90.000,E1 30.463} C_DIS
LIN {X -0.045,Y -189.149,Z 1116.151,A 0.000,B 0.000,C 90.000,E1 27.206} C_DIS
LIN {X -0.064,Y -184.412,Z 1116.133,A 0.000,B 0.000,C 90.000,E1 23.898} C_DIS
LIN {X -0.083,Y -180.336,Z 1116.114,A 0.000,B 0.000,C 90.000,E1 20.556} C_DIS
LIN {X -0.044,Y -176.207,Z 1116.091,A 0.000,B 0.000,C 90.000,E1 16.315} C_DIS
LIN {X 0.081,Y -173.081,Z 1116.067,A 0.000,B 0.000,C 90.000,E1 12.007} C_DIS
LIN {X -0.052,Y -170.500,Z 1116.033,A 0.000,B 0.000,C 90.000,E1 6.030} C_DIS
LIN {X 0.072,Y -171.343,Z 1115.964,A 0.000,B 0.000,C 90.000,E1 353.457} C_DIS
LIN {X -0.073,Y -174.073,Z 1115.935,A 0.000,B 0.000,C 90.000,E1 348.342} C_DIS
LIN {X 0.034,Y -177.470,Z 1115.911,A 0.000,B 0.000,C 90.000,E1 344.031} C_DIS
LIN {X -0.077,Y -181.699,Z 1115.888,A 0.000,B 0.000,C 90.000,E1 339.826} C_DIS
LIN {X 0.022,Y -185.809,Z 1115.869,A 0.000,B 0.000,C 90.000,E1 336.433} C_DIS
LIN {X -0.057,Y -190.634,Z 1115.851,A 0.000,B 0.000,C 90.000,E1 333.127} C_DIS
LIN {X 0.083,Y -196.153,Z 1115.832,A 0.000,B 0.000,C 90.000,E1 329.793} C_DIS
LIN {X -0.053,Y -202.342,Z 1115.814,A 0.000,B 0.000,C 90.000,E1 326.580} C_DIS
LIN {X 0.077,Y -209.350,Z 1115.796,A 0.000,B 0.000,C 90.000,E1 323.336} C_DIS
LIN {X -0.070,Y -218.098,Z 1115.777,A 0.000,B 0.000,C 90.000,E1 319.828} C_DIS
LIN {X 0.063,Y -226.835,Z 1115.760,A 0.000,B 0.000,C 90.000,E1 316.701} C_DIS
LIN {X -0.087,Y -236.592,Z 1115.743,A 0.000,B 0.000,C 90.000,E1 313.704} C_DIS
LIN {X 0.038,Y -247.596,Z 1115.726,A 0.000,B 0.000,C 90.000,E1 310.701} C_DIS
LIN {X -0.063,Y -258.511,Z 1115.712,A 0.000,B 0.000,C 90.000,E1 308.177} C_DIS
LIN {X -0.034,Y -274.257,Z 1115.694,A 0.000,B 0.000,C 90.000,E1 304.978} C_DIS
LIN {X -0.018,Y -291.232,Z 1115.677,A 0.000,B 0.000,C 90.000,E1 301.878} C_DIS
LIN {X -0.022,Y -305.695,Z 1115.664,A 0.000,B 0.000,C 90.000,E1 299.539} C_DIS
LIN {X -0.007,Y -325.958,Z 1115.648,A 0.000,B 0.000,C 90.000,E1 296.616} C_DIS
LIN {X 0.203,Y -343.257,Z 1115.636,A 0.000,B 0.000,C 90.000,E1 294.387} C_DIS
LIN {X -0.028,Y -356.293,Z 1115.627,A 0.000,B 0.000,C 90.000,E1 292.950} C_DIS
LIN {X -0.090,Y -372.381,Z 1115.618,A 0.000,B 0.000,C 90.000,E1 291.334} C_DIS
LIN {X -0.235,Y -394.056,Z 1115.608,A 0.000,B 0.000,C 90.000,E1 289.396} C_DIS
LIN {X -0.219,Y -407.604,Z 1115.601,A 0.000,B 0.000,C 90.000,E1 288.181} C_DIS
LIN {X 0.036,Y -418.202,Z 1115.595,A 0.000,B 0.000,C 90.000,E1 287.166} C_DIS
LIN {X -0.157,Y -428.258,Z 1115.590,A 0.000,B 0.000,C 90.000,E1 286.205} C_DIS
LIN {X -0.131,Y -435.612,Z 1115.586,A 0.000,B 0.000,C 90.000,E1 285.426} C_DIS
LIN {X -0.079,Y -444.941,Z 1115.580,A 0.000,B 0.000,C 90.000,E1 284.356} C_DIS
LIN {X 0.173,Y -451.261,Z 1115.575,A 0.000,B 0.000,C 90.000,E1 283.536} C_DIS
LIN {X 0.044,Y -456.870,Z 1115.571,A 0.000,B 0.000,C 90.000,E1 282.771} C_DIS
LIN {X -0.034,Y -461.762,Z 1115.567,A 0.000,B 0.000,C 90.000,E1 282.007} C_DIS
LIN {X -0.077,Y -465.989,Z 1115.562,A 0.000,B 0.000,C 90.000,E1 281.243} C_DIS
LIN {X -0.169,Y -469.636,Z 1115.558,A 0.000,B 0.000,C 90.000,E1 280.489} C_DIS
LIN {X -0.148,Y -472.704,Z 1115.554,A 0.000,B 0.000,C 90.000,E1 279.726} C_DIS
LIN {X -0.048,Y -474.434,Z 1115.551,A 0.000,B 0.000,C 90.000,E1 279.208} C_DIS
LIN {X 0.069,Y -475.898,Z 1115.548,A 0.000,B 0.000,C 90.000,E1 278.690} C_DIS
LIN {X -0.206,Y -477.072,Z 1115.546,A 0.000,B 0.000,C 90.000,E1 278.219} C_DIS
LIN {X -0.070,Y -477.976,Z 1115.543,A 0.000,B 0.000,C 90.000,E1 277.701} C_DIS
LIN {X 0.075,Y -478.561,Z 1115.540,A 0.000,B 0.000,C 90.000,E1 277.182} C_DIS
LIN {X 0.226,Y -478.929,Z 1115.537,A 0.000,B 0.000,C 90.000,E1 276.663} C_DIS
LIN {X -0.095,Y -478.960,Z 1115.534,A 0.000,B 0.000,C 90.000,E1 276.201} C_DIS
LIN {X 0.061,Y -478.608,Z 1115.532,A 0.000,B 0.000,C 90.000,E1 275.682} C_DIS
LIN {X 0.216,Y -477.952,Z 1115.529,A 0.000,B 0.000,C 90.000,E1 275.163} C_DIS
LIN {X -0.108,Y -476.972,Z 1115.526,A 0.000,B 0.000,C 90.000,E1 274.702} C_DIS
LIN {X 0.002,Y -475.529,Z 1115.523,A 0.000,B 0.000,C 90.000,E1 274.188} C_DIS
LIN {X 0.142,Y -473.573,Z 1115.521,A 0.000,B 0.000,C 90.000,E1 273.669} C_DIS
LIN {X -0.228,Y -470.967,Z 1115.518,A 0.000,B 0.000,C 90.000,E1 273.212} C_DIS
LIN {X -0.117,Y -467.583,Z 1115.515,A 0.000,B 0.000,C 90.000,E1 272.694} C_DIS
LIN {X -0.048,Y -463.134,Z 1115.512,A 0.000,B 0.000,C 90.000,E1 272.178} C_DIS
LIN {X 0.015,Y -457.450,Z 1115.509,A 0.000,B 0.000,C 90.000,E1 271.661} C_DIS
LIN {X 0.083,Y -451.046,Z 1115.507,A 0.000,B 0.000,C 90.000,E1 271.203} C_DIS
LIN {X -0.187,Y -444.242,Z 1115.505,A 0.000,B 0.000,C 90.000,E1 270.859} C_DIS
LIN {X 0.067,Y -437.342,Z 1115.503,A 0.000,B 0.000,C 90.000,E1 270.516} C_DIS
LIN {X -0.156,Y -430.165,Z 1115.501,A 0.000,B 0.000,C 90.000,E1 270.286} C_DIS
LIN {X -0.046,Y -423.114,Z 1115.500,A 0.000,B 0.000,C 90.000,E1 270.057} C_DIS
LIN {X -0.116,Y -415.670,Z 1115.499,A 0.000,B 0.000,C 90.000,E1 269.885} C_DIS
LIN {X 0.041,Y -407.705,Z 1115.498,A 0.000,B 0.000,C 90.000,E1 269.714} C_DIS
LIN {X 0.028,Y -398.201,Z 1115.498,A 0.000,B 0.000,C 90.000,E1 269.599} C_DIS
LIN {X -0.004,Y -386.182,Z 1115.497,A 0.000,B 0.000,C 90.000,E1 269.542} C_DIS
LIN {X -0.034,Y -181.446,Z 1115.497,A 0.000,B 0.000,C 90.000,E1 269.542} C_DIS
LIN {X 0.089,Y -180.857,Z 1115.472,A 0.000,B 0.000,C 90.000,E1 264.951} C_DIS
LIN {X -0.037,Y -178.969,Z 1115.444,A 0.000,B 0.000,C 90.000,E1 259.926} C_DIS
LIN {X -0.027,Y -177.924,Z 1115.435,A 0.000,B 0.000,C 90.000,E1 258.229} C_DIS
LIN {X -0.012,Y -175.562,Z 1115.411,A 0.000,B 0.000,C 90.000,E1 253.976} C_DIS
LIN {X -0.005,Y -172.291,Z 1115.387,A 0.000,B 0.000,C 90.000,E1 249.699} C_DIS
LIN {X -0.027,Y -171.769,Z 1115.382,A 0.000,B 0.000,C 90.000,E1 248.847} C_DIS
LIN {X -0.035,Y -168.011,Z 1115.359,A 0.000,B 0.000,C 90.000,E1 244.537} C_DIS
LIN {X -0.016,Y -166.761,Z 1115.349,A 0.000,B 0.000,C 90.000,E1 242.794} C_DIS
LIN {X 0.043,Y -162.741,Z 1115.325,A 0.000,B 0.000,C 90.000,E1 238.408} C_DIS
LIN {X 0.105,Y -161.431,Z 1115.315,A 0.000,B 0.000,C 90.000,E1 236.628} C_DIS
LIN {X -0.076,Y -157.424,Z 1115.290,A 0.000,B 0.000,C 90.000,E1 232.271} C_DIS
LIN {X 0.077,Y -155.428,Z 1115.275,A 0.000,B 0.000,C 90.000,E1 229.542} C_DIS
LIN {X 0.007,Y -151.752,Z 1115.250,A 0.000,B 0.000,C 90.000,E1 225.081} C_DIS
LIN {X 0.019,Y -149.952,Z 1115.235,A 0.000,B 0.000,C 90.000,E1 222.366} C_DIS
LIN {X 0.047,Y -146.795,Z 1115.210,A 0.000,B 0.000,C 90.000,E1 217.810} C_DIS
LIN {X -0.053,Y -145.370,Z 1115.195,A 0.000,B 0.000,C 90.000,E1 215.105} C_DIS
LIN {X 0.063,Y -142.434,Z 1115.164,A 0.000,B 0.000,C 90.000,E1 209.539} C_DIS
LIN {X -0.014,Y -141.425,Z 1115.149,A 0.000,B 0.000,C 90.000,E1 206.796} C_DIS
LIN {X -0.032,Y -139.363,Z 1115.113,A 0.000,B 0.000,C 90.000,E1 200.301} C_DIS
LIN {X -0.045,Y -138.808,Z 1115.097,A 0.000,B 0.000,C 90.000,E1 197.511} C_DIS
LIN {X 0.005,Y -138.350,Z 1115.056,A 0.000,B 0.000,C 90.000,E1 190.018} C_DIS
LIN {X -0.019,Y -139.543,Z 1115.004,A 0.000,B 0.000,C 90.000,E1 180.688} C_DIS
LIN {X 0.074,Y -141.242,Z 1114.973,A 0.000,B 0.000,C 90.000,E1 175.065} C_DIS
LIN {X 0.033,Y -142.612,Z 1114.957,A 0.000,B 0.000,C 90.000,E1 172.299} C_DIS
LIN {X -0.014,Y -144.926,Z 1114.932,A 0.000,B 0.000,C 90.000,E1 167.701} C_DIS
LIN {X -0.022,Y -147.554,Z 1114.911,A 0.000,B 0.000,C 90.000,E1 164.031} C_DIS
LIN {X 0.009,Y -150.158,Z 1114.891,A 0.000,B 0.000,C 90.000,E1 160.369} C_DIS
LIN {X 0.018,Y -153.531,Z 1114.871,A 0.000,B 0.000,C 90.000,E1 156.741} C_DIS
LIN {X 0.072,Y -156.949,Z 1114.851,A 0.000,B 0.000,C 90.000,E1 153.127} C_DIS
LIN {X 0.008,Y -161.054,Z 1114.831,A 0.000,B 0.000,C 90.000,E1 149.587} C_DIS
LIN {X 0.092,Y -163.162,Z 1114.821,A 0.000,B 0.000,C 90.000,E1 147.788} C_DIS
LIN {X -0.037,Y -167.581,Z 1114.802,A 0.000,B 0.000,C 90.000,E1 144.322} C_DIS
LIN {X 0.009,Y -171.410,Z 1114.787,A 0.000,B 0.000,C 90.000,E1 141.698} C_DIS
LIN {X 0.048,Y -176.326,Z 1114.768,A 0.000,B 0.000,C 90.000,E1 138.243} C_DIS
LIN {X -0.084,Y -180.615,Z 1114.754,A 0.000,B 0.000,C 90.000,E1 135.729} C_DIS
LIN {X 0.030,Y -186.016,Z 1114.735,A 0.000,B 0.000,C 90.000,E1 132.324} C_DIS
LIN {X -0.052,Y -190.651,Z 1114.721,A 0.000,B 0.000,C 90.000,E1 129.850} C_DIS
LIN {X 0.011,Y -196.402,Z 1114.703,A 0.000,B 0.000,C 90.000,E1 126.537} C_DIS
LIN {X -0.085,Y -200.454,Z 1114.692,A 0.000,B 0.000,C 90.000,E1 124.532} C_DIS
LIN {X 0.090,Y -308.784,Z 1114.692,A 0.000,B 0.000,C 90.000,E1 124.485} C_DIS
LIN {X -0.012,Y -310.074,Z 1114.692,A 0.000,B 0.000,C 90.000,E1 124.485} C_DIS
LIN {X 0.069,Y -314.625,Z 1114.691,A 0.000,B 0.000,C 90.000,E1 124.278} C_DIS
LIN {X -0.111,Y -317.076,Z 1114.689,A 0.000,B 0.000,C 90.000,E1 124.119} C_DIS
LIN {X 0.069,Y -320.904,Z 1114.687,A 0.000,B 0.000,C 90.000,E1 123.627} C_DIS
LIN {X 0.150,Y -322.745,Z 1114.685,A 0.000,B 0.000,C 90.000,E1 123.293} C_DIS
LIN {X -0.040,Y -324.178,Z 1114.683,A 0.000,B 0.000,C 90.000,E1 123.007} C_DIS
LIN {X -0.144,Y -336.006,Z 1114.666,A 0.000,B 0.000,C 90.000,E1 119.873} C_DIS
LIN {X -0.060,Y -348.049,Z 1114.650,A 0.000,B 0.000,C 90.000,E1 117.078} C_DIS
LIN {X 0.056,Y -361.567,Z 1114.635,A 0.000,B 0.000,C 90.000,E1 114.335} C_DIS
LIN {X 0.016,Y -374.912,Z 1114.622,A 0.000,B 0.000,C 90.000,E1 111.972} C_DIS
LIN {X 0.170,Y -389.607,Z 1114.609,A 0.000,B 0.000,C 90.000,E1 109.631} C_DIS
LIN {X -0.076,Y -405.757,Z 1114.597,A 0.000,B 0.000,C 90.000,E1 107.402} C_DIS
LIN {X -0.051,Y -423.474,Z 1114.584,A 0.000,B 0.000,C 90.000,E1 105.190} C_DIS
LIN {X -0.179,Y -442.824,Z 1114.572,A 0.000,B 0.000,C 90.000,E1 103.063} C_DIS
LIN {X -0.199,Y -463.013,Z 1114.561,A 0.000,B 0.000,C 90.000,E1 101.074} C_DIS
LIN {X -0.200,Y -468.133,Z 1114.559,A 0.000,B 0.000,C 90.000,E1 100.602} C_DIS
LIN {X -0.195,Y -470.246,Z 1114.557,A 0.000,B 0.000,C 90.000,E1 100.366} C_DIS
LIN {X 0.191,Y -471.845,Z 1114.556,A 0.000,B 0.000,C 90.000,E1 100.084} C_DIS
LIN {X 0.049,Y -473.154,Z 1114.555,A 0.000,B 0.000,C 90.000,E1 99.849} C_DIS
LIN {X -0.096,Y -474.120,Z 1114.553,A 0.000,B 0.000,C 90.000,E1 99.613} C_DIS
LIN {X 0.020,Y -475.201,Z 1114.551,A 0.000,B 0.000,C 90.000,E1 99.095} C_DIS
LIN {X 0.217,Y -475.291,Z 1114.548,A 0.000,B 0.000,C 90.000,E1 98.568} C_DIS
LIN {X -0.122,Y -474.408,Z 1114.545,A 0.000,B 0.000,C 90.000,E1 98.106} C_DIS
LIN {X 0.010,Y -472.405,Z 1114.542,A 0.000,B 0.000,C 90.000,E1 97.587} C_DIS
LIN {X -0.128,Y -470.858,Z 1114.541,A 0.000,B 0.000,C 90.000,E1 97.352} C_DIS
LIN {X 0.207,Y -456.369,Z 1114.529,A 0.000,B 0.000,C 90.000,E1 95.277} C_DIS
LIN {X -0.101,Y -440.492,Z 1114.516,A 0.000,B 0.000,C 90.000,E1 92.980} C_DIS
LIN {X -0.107,Y -427.448,Z 1114.505,A 0.000,B 0.000,C 90.000,E1 90.859} C_DIS
LIN {X 0.204,Y -412.124,Z 1114.490,A 0.000,B 0.000,C 90.000,E1 88.108} C_DIS
LIN {X -0.145,Y -403.185,Z 1114.480,A 0.000,B 0.000,C 90.000,E1 86.502} C_DIS
LIN {X 0.170,Y -394.115,Z 1114.471,A 0.000,B 0.000,C 90.000,E1 84.780} C_DIS
LIN {X -0.019,Y -382.059,Z 1114.458,A 0.000,B 0.000,C 90.000,E1 82.534} C_DIS
LIN {X 0.038,Y -372.963,Z 1114.449,A 0.000,B 0.000,C 90.000,E1 80.792} C_DIS
LIN {X -0.048,Y -365.096,Z 1114.441,A 0.000,B 0.000,C 90.000,E1 79.342} C_DIS
LIN {X 0.198,Y -355.331,Z 1114.431,A 0.000,B 0.000,C 90.000,E1 77.521} C_DIS
LIN {X -0.148,Y -343.762,Z 1114.419,A 0.000,B 0.000,C 90.000,E1 75.463} C_DIS
LIN {X 0.066,Y -330.639,Z 1114.405,A 0.000,B 0.000,C 90.000,E1 72.960} C_DIS
LIN {X -0.083,Y -315.066,Z 1114.388,A 0.000,B 0.000,C 90.000,E1 69.826} C_DIS
LIN {X -0.154,Y -301.913,Z 1114.372,A 0.000,B 0.000,C 90.000,E1 66.922} C_DIS
LIN {X 0.063,Y -290.744,Z 1114.357,A 0.000,B 0.000,C 90.000,E1 64.229} C_DIS
LIN {X 0.112,Y -279.930,Z 1114.342,A 0.000,B 0.000,C 90.000,E1 61.513} C_DIS
LIN {X -0.003,Y -270.755,Z 1114.328,A 0.000,B 0.000,C 90.000,E1 59.125} C_DIS
LIN {X 0.000,Y -259.252,Z 1114.311,A 0.000,B 0.000,C 90.000,E1 55.960} C_DIS
LIN {X 0.042,Y -248.467,Z 1114.293,A 0.000,B 0.000,C 90.000,E1 52.718} C_DIS
LIN {X 0.049,Y -239.385,Z 1114.277,A 0.000,B 0.000,C 90.000,E1 49.784} C_DIS
LIN {X -0.035,Y -231.019,Z 1114.260,A 0.000,B 0.000,C 90.000,E1 46.824} C_DIS
LIN {X 0.005,Y -223.106,Z 1114.243,A 0.000,B 0.000,C 90.000,E1 43.785} C_DIS
LIN {X 0.020,Y -215.527,Z 1114.226,A 0.000,B 0.000,C 90.000,E1 40.701} C_DIS
LIN {X 0.029,Y -208.334,Z 1114.209,A 0.000,B 0.000,C 90.000,E1 37.569} C_DIS
LIN {X 0.065,Y -200.051,Z 1114.187,A 0.000,B 0.000,C 90.000,E1 33.579} C_DIS
LIN {X 0.093,Y -194.104,Z 1114.169,A 0.000,B 0.000,C 90.000,E1 30.335} C_DIS
LIN {X 0.024,Y -188.710,Z 1114.151,A 0.000,B 0.000,C 90.000,E1 27.078} C_DIS
LIN {X -0.007,Y -183.988,Z 1114.132,A 0.000,B 0.000,C 90.000,E1 23.770} C_DIS
LIN {X -0.040,Y -179.958,Z 1114.113,A 0.000,B 0.000,C 90.000,E1 20.429} C_DIS
LIN {X -0.067,Y -175.851,Z 1114.090,A 0.000,B 0.000,C 90.000,E1 16.205} C_DIS
LIN {X 0.054,Y -172.731,Z 1114.066,A 0.000,B 0.000,C 90.000,E1 11.895} C_DIS
LIN {X -0.069,Y -170.214,Z 1114.033,A 0.000,B 0.000,C 90.000,E1 5.910} C_DIS
LIN {X 0.062,Y -171.072,Z 1113.964,A 0.000,B 0.000,C 90.000,E1 353.457} C_DIS
LIN {X 0.076,Y -173.783,Z 1113.935,A 0.000,B 0.000,C 90.000,E1 348.285} C_DIS
LIN {X 0.003,Y -177.140,Z 1113.911,A 0.000,B 0.000,C 90.000,E1 344.031} C_DIS
LIN {X -0.057,Y -181.389,Z 1113.888,A 0.000,B 0.000,C 90.000,E1 339.806} C_DIS
LIN {X -0.081,Y -186.639,Z 1113.864,A 0.000,B 0.000,C 90.000,E1 335.613} C_DIS
LIN {X -0.057,Y -191.665,Z 1113.846,A 0.000,B 0.000,C 90.000,E1 332.281} C_DIS
LIN {X -0.060,Y -197.365,Z 1113.828,A 0.000,B 0.000,C 90.000,E1 328.997} C_DIS
LIN {X 0.051,Y -203.800,Z 1113.810,A 0.000,B 0.000,C 90.000,E1 325.722} C_DIS
LIN {X -0.067,Y -211.002,Z 1113.792,A 0.000,B 0.000,C 90.000,E1 322.557} C_DIS
LIN {X 0.053,Y -218.947,Z 1113.774,A 0.000,B 0.000,C 90.000,E1 319.380} C_DIS
LIN {X 0.043,Y -227.792,Z 1113.757,A 0.000,B 0.000,C 90.000,E1 316.296} C_DIS
LIN {X -0.082,Y -237.764,Z 1113.740,A 0.000,B 0.000,C 90.000,E1 313.299} C_DIS
LIN {X -0.086,Y -247.475,Z 1113.726,A 0.000,B 0.000,C 90.000,E1 310.701} C_DIS
LIN {X 0.168,Y -258.424,Z 1113.712,A 0.000,B 0.000,C 90.000,E1 308.096} C_DIS
LIN {X -0.019,Y -274.207,Z 1113.694,A 0.000,B 0.000,C 90.000,E1 304.945} C_DIS
LIN {X -0.169,Y -291.276,Z 1113.677,A 0.000,B 0.000,C 90.000,E1 301.878} C_DIS
LIN {X 0.086,Y -305.763,Z 1113.664,A 0.000,B 0.000,C 90.000,E1 299.489} C_DIS
LIN {X -0.174,Y -326.062,Z 1113.648,A 0.000,B 0.000,C 90.000,E1 296.616} C_DIS
LIN {X 0.050,Y -343.352,Z 1113.635,A 0.000,B 0.000,C 90.000,E1 294.387} C_DIS
LIN {X 0.134,Y -356.415,Z 1113.627,A 0.000,B 0.000,C 90.000,E1 292.898} C_DIS
LIN {X 0.025,Y -369.919,Z 1113.620,A 0.000,B 0.000,C 90.000,E1 291.535} C_DIS
LIN {X 0.088,Y -391.968,Z 1113.609,A 0.000,B 0.000,C 90.000,E1 289.523} C_DIS
LIN {X -0.176,Y -405.418,Z 1113.602,A 0.000,B 0.000,C 90.000,E1 288.362} C_DIS
LIN {X -0.249,Y -416.028,Z 1113.596,A 0.000,B 0.000,C 90.000,E1 287.402} C_DIS
LIN {X 0.018,Y -426.150,Z 1113.591,A 0.000,B 0.000,C 90.000,E1 286.386} C_DIS
LIN {X 0.059,Y -433.703,Z 1113.587,A 0.000,B 0.000,C 90.000,E1 285.607} C_DIS
LIN {X -0.063,Y -440.886,Z 1113.582,A 0.000,B 0.000,C 90.000,E1 284.828} C_DIS
LIN {X 0.151,Y -447.605,Z 1113.578,A 0.000,B 0.000,C 90.000,E1 284.008} C_DIS
LIN {X -0.011,Y -453.696,Z 1113.574,A 0.000,B 0.000,C 90.000,E1 283.244} C_DIS
LIN {X -0.116,Y -459.002,Z 1113.569,A 0.000,B 0.000,C 90.000,E1 282.479} C_DIS
LIN {X -0.182,Y -463.667,Z 1113.565,A 0.000,B 0.000,C 90.000,E1 281.715} C_DIS
LIN {X -0.205,Y -467.675,Z 1113.561,A 0.000,B 0.000,C 90.000,E1 280.950} C_DIS
LIN {X 0.178,Y -471.131,Z 1113.557,A 0.000,B 0.000,C 90.000,E1 280.141} C_DIS
LIN {X -0.111,Y -473.059,Z 1113.554,A 0.000,B 0.000,C 90.000,E1 279.670} C_DIS
LIN {X -0.007,Y -474.729,Z 1113.551,A 0.000,B 0.000,C 90.000,E1 279.151} C_DIS
LIN {X 0.184,Y -476.189,Z 1113.548,A 0.000,B 0.000,C 90.000,E1 278.624} C_DIS
LIN {X -0.161,Y -477.366,Z 1113.545,A 0.000,B 0.000,C 90.000,E1 278.163} C_DIS
LIN {X -0.022,Y -478.252,Z 1113.542,A 0.000,B 0.000,C 90.000,E1 277.644} C_DIS
LIN {X 0.125,Y -478.821,Z 1113.540,A 0.000,B 0.000,C 90.000,E1 277.125} C_DIS
LIN {X -0.198,Y -479.160,Z 1113.537,A 0.000,B 0.000,C 90.000,E1 276.663} C_DIS
LIN {X -0.041,Y -479.174,Z 1113.534,A 0.000,B 0.000,C 90.000,E1 276.144} C_DIS
LIN {X 0.117,Y -478.832,Z 1113.531,A 0.000,B 0.000,C 90.000,E1 275.625} C_DIS
LIN {X -0.202,Y -478.189,Z 1113.529,A 0.000,B 0.000,C 90.000,E1 275.163} C_DIS
LIN {X -0.049,Y -477.148,Z 1113.526,A 0.000,B 0.000,C 90.000,E1 274.645} C_DIS
LIN {X 0.063,Y -475.699,Z 1113.523,A 0.000,B 0.000,C 90.000,E1 274.131} C_DIS
LIN {X 0.204,Y -473.699,Z 1113.520,A 0.000,B 0.000,C 90.000,E1 273.612} C_DIS
END
